// TIA Portal V18 program export: 17 tag tables, 0 data types, 18 data blocks, 24 code blocks (in call order from the OBs), 7 instance data blocks

VAR_GLOBAL   // PLC tag table "PLC_Simulation_Tags"
   "1400_FT115_PV" AT %MD100 : Real;   // Lưu lượng dòng liệu đo được tại FT115
   "1400_FT101_PV" AT %MD104 : Real;   // Lưu lượng dòng liệu đo được tại FT101
   "1400_1_02_PV" AT %MD108 : Real;   // Giá trị đo của cảm biến 1-02
   "1406_TX35_PV" AT %MD112 : Real;   // Giá trị đo cảm biến nhiệt độ/áp suất TX35
   "1400_TT64_PV" AT %MD116 : Real;   // Nhiệt độ đo được tại TT64
   "1400_TT32_PV" AT %MD120 : Real;   // Nhiệt độ đo được tại TT32
   "1400_LGFE01_PV" AT %MD124 : Real;   // Mức bồn hoặc lưu lượng đo tại LGFE01
   "1400_FS51_PV" AT %MD128 : Real;   // Giá trị lưu lượng đo được tại FS51
   "1400_FY301_PV" AT %MD132 : Real;   // Mức cân hoặc vị trí điều khiển bồn FY301
   "1400_TT101_PV" AT %MD136 : Real;   // Nhiệt độ đo được tại TT101
   "1400_FTT02_PV" AT %MD140 : Real;   // Lưu lượng/nhiệt độ đo được tại FTT02
   "1500S_Trang_Thai" AT %M200.0 : Bool;   // Trạng thái hoạt động dòng liệu 1500S (0: Không chảy, 1: Đang chảy)
   "1404T_Trang_Thai" AT %M200.1 : Bool;   // Trạng thái hoạt động dòng liệu 1404T
   CR_2013_FO_104_Trang_Thai AT %M200.2 : Bool;   // Trạng thái hoạt động dòng liệu CR-2013-FO-104
   BFOC_SS_20_06_Trang_Thai AT %M200.3 : Bool;   // Trạng thái hoạt động dòng liệu BFOC-SS-20-06
   PC03010T01_Trang_Thai AT %M200.4 : Bool;   // Trạng thái dòng liệu đầu ra PC03010T01
   "1401_Trang_Thai" AT %M200.5 : Bool;   // Trạng thái dòng liệu xả đáy 1401
   "1400_PT91_Chay" AT %M200.6 : Bool;   // Tín hiệu báo chạy bơm 1400PT91 (1: Chạy)
   "1400_KCK01_Chay" AT %M200.7 : Bool;   // Tín hiệu báo chạy cánh khuấy bồn 1400KCK01
   "1400_FT102_Mo" AT %M201.0 : Bool;   // Tín hiệu báo mở van nạp liệu 1400FT102
   "1400_TY33_Mo" AT %M201.1 : Bool;   // Tín hiệu báo mở van điều khiển cooling 1400TY33
   "160_FEC53_Mo" AT %M201.2 : Bool;   // Tín hiệu báo mở van kẹp 160 FEC53
   "1400_TXC32_Mo" AT %M201.3 : Bool;   // Tín hiệu báo mở van điều khiển 1400TXC32
   "1400_TC32_Mo" AT %M201.4 : Bool;   // Tín hiệu báo mở van điều khiển 1400TC32
   "1400_FIC01_Mo" AT %M201.5 : Bool;   // Tín hiệu báo mở van điều khiển 1400FIC01
   "1400_FS51_Mo" AT %M201.6 : Bool;   // Tín hiệu báo mở van xả đáy 1400FS51
   "1500S_Status" AT %MW300 : Int;   // Mã trạng thái dòng liệu 1500S (0: Dừng, 1: Chạy, 2: Lỗi)
   "1404T_Status" AT %MW302 : Int;   // Mã trạng thái dòng liệu 1404T
   CR_2013_FO_104_Status AT %MW304 : Int;   // Mã trạng thái dòng liệu CR-2013-FO-104
   BFOC_SS_20_06_Status AT %MW306 : Int;   // Mã trạng thái dòng liệu BFOC-SS-20-06
   PC03010T01_Status AT %MW308 : Int;   // Mã trạng thái dòng liệu PC03010T01
   "1401_Status" AT %MW310 : Int;   // Mã trạng thái dòng liệu xả đáy 1401
   "1400_PT91_Status" AT %MW312 : Int;   // Mã trạng thái hoạt động bơm 1400PT91 (0: Dừng, 1: Chạy, 2: Lỗi)
   "1400_KCK01_Status" AT %MW314 : Int;   // Mã trạng thái hoạt động cánh khuấy 1400KCK01
   "1400_FT102_Status" AT %MW316 : Int;   // Mã trạng thái hoạt động van 1400FT102 (0: Đóng, 1: Mở, 2: Lỗi)
   "1400_TY33_Status" AT %MW318 : Int;   // Mã trạng thái hoạt động van 1400TY33
   "160_FEC53_Status" AT %MW320 : Int;   // Mã trạng thái hoạt động van 160 FEC53
   "1400_TXC32_Status" AT %MW322 : Int;   // Mã trạng thái hoạt động van 1400TXC32
   "1400_TC32_Status" AT %MW324 : Int;   // Mã trạng thái hoạt động van 1400TC32
   "1400_FIC01_Status" AT %MW326 : Int;   // Mã trạng thái hoạt động van 1400FIC01
   "1400_FS51_Status" AT %MW328 : Int;   // Mã trạng thái hoạt động van 1400FS51
   Sim_Counter AT %MD400 : Real;   // Biến đếm trung gian cho sóng tam giác mô phỏng
   Sim_Dir AT %M404.0 : Bool;   // Bit hướng đếm mô phỏng (0: Tăng, 1: Giảm)
   Sim_Val_Norm AT %MD408 : Real;   // Giá trị đếm đã chuẩn hóa về dải 0.0 - 1.0
   Timer_Sim_Pulse_Output AT %M404.1 : Bool;   // Xung kích hoạt đếm từ Timer
END_VAR

VAR_GLOBAL   // PLC tag table "AI_Tags"
   AI_Nut_Khoi_Dong AT %I0.0 : Bool;   // Nút khởi động vật lý
   AI_Nut_Khoi_Dong_HMI AT %M110.0 : Bool;   // Tín hiệu mô phỏng/HMI song song cho Nút khởi động vật lý
   AI_Nut_Khoi_Dong_HMI_Gated AT %M320.0 : Bool;   // Tín hiệu HMI đã qua xử lý chế độ cho Nút khởi động vật lý
   AI_Nut_Khoi_Dong_Eff AT %M320.1 : Bool;   // Tín hiệu thực tế/mô phỏng hiệu dụng cho Nút khởi động vật lý
   AI_Nut_Dung AT %I0.1 : Bool;   // Nút dừng vật lý
   AI_Nut_Dung_HMI AT %M110.1 : Bool;   // Tín hiệu mô phỏng/HMI song song cho Nút dừng vật lý
   AI_Nut_Dung_HMI_Gated AT %M320.2 : Bool;   // Tín hiệu HMI đã qua xử lý chế độ cho Nút dừng vật lý
   AI_Nut_Dung_Eff AT %M320.3 : Bool;   // Tín hiệu thực tế/mô phỏng hiệu dụng cho Nút dừng vật lý
   AI_Nut_Reset AT %I0.2 : Bool;   // Nút reset lỗi vật lý
   AI_Nut_Reset_HMI AT %M110.2 : Bool;   // Tín hiệu mô phỏng/HMI song song cho Nút reset lỗi vật lý
   AI_Nut_Reset_HMI_Gated AT %M320.4 : Bool;   // Tín hiệu HMI đã qua xử lý chế độ cho Nút reset lỗi vật lý
   AI_Nut_Reset_Eff AT %M320.5 : Bool;   // Tín hiệu thực tế/mô phỏng hiệu dụng cho Nút reset lỗi vật lý
   AI_Nut_EStop AT %I0.3 : Bool;   // Nút dừng khẩn vật lý
   AI_Nut_EStop_HMI AT %M110.3 : Bool;   // Tín hiệu mô phỏng/HMI song song cho Nút dừng khẩn vật lý
   AI_Nut_EStop_HMI_Gated AT %M320.6 : Bool;   // Tín hiệu HMI đã qua xử lý chế độ cho Nút dừng khẩn vật lý
   AI_Nut_EStop_Eff AT %M320.7 : Bool;   // Tín hiệu thực tế/mô phỏng hiệu dụng cho Nút dừng khẩn vật lý
   AI_FT3200_Bon1 AT %ID100 : Real;   // Cảm biến lưu lượng nước dosing vào Bồn 1
   AI_FT3200_Bon1_HMI AT %MD700 : Real;   // Giá trị mô phỏng/HMI song song cho Cảm biến lưu lượng nước dosing vào Bồn 1
   AI_FT3200_Bon1_Use_HMI AT %M420.0 : Bool;   // Chọn chế độ mô phỏng HMI cho Cảm biến lưu lượng nước dosing vào Bồn 1
   AI_FT3200_Bon1_Sim_Req AT %M321.0 : Bool;   // Yêu cầu mô phỏng cảm biến cho Cảm biến lưu lượng nước dosing vào Bồn 1
   AI_FT3200_Bon1_Sim_Active AT %M321.1 : Bool;   // Mô phỏng cảm biến đang hoạt động cho Cảm biến lưu lượng nước dosing vào Bồn 1
   AI_FT3200_Bon1_Eff AT %MD704 : Real;   // Giá trị thực tế/mô phỏng hiệu dụng cho Cảm biến lưu lượng nước dosing vào Bồn 1
   AI_FQ3200_Bon1 AT %ID104 : Real;   // Bộ đếm lưu lượng tích lũy Bồn 1
   AI_FQ3200_Bon1_HMI AT %MD708 : Real;   // Giá trị mô phỏng/HMI song song cho Bộ đếm lưu lượng tích lũy Bồn 1
   AI_FQ3200_Bon1_Use_HMI AT %M420.1 : Bool;   // Chọn chế độ mô phỏng HMI cho Bộ đếm lưu lượng tích lũy Bồn 1
   AI_FQ3200_Bon1_Sim_Req AT %M321.2 : Bool;   // Yêu cầu mô phỏng cảm biến cho Bộ đếm lưu lượng tích lũy Bồn 1
   AI_FQ3200_Bon1_Sim_Active AT %M321.3 : Bool;   // Mô phỏng cảm biến đang hoạt động cho Bộ đếm lưu lượng tích lũy Bồn 1
   AI_FQ3200_Bon1_Eff AT %MD712 : Real;   // Giá trị thực tế/mô phỏng hiệu dụng cho Bộ đếm lưu lượng tích lũy Bồn 1
   AI_LS3202_Bon1_Cao AT %I0.4 : Bool;   // Cảm biến mức cao Bồn 1
   AI_LS3202_Bon1_Cao_HMI AT %M110.4 : Bool;   // Tín hiệu mô phỏng/HMI song song cho Cảm biến mức cao Bồn 1
   AI_LS3202_Bon1_Cao_HMI_Gated AT %M321.4 : Bool;   // Tín hiệu HMI đã qua xử lý chế độ cho Cảm biến mức cao Bồn 1
   AI_LS3202_Bon1_Cao_Eff AT %M321.5 : Bool;   // Tín hiệu thực tế/mô phỏng hiệu dụng cho Cảm biến mức cao Bồn 1
   AI_LT3203_Bon1 AT %ID108 : Real;   // Cảm biến mức liên tục Bồn 1
   AI_LT3203_Bon1_HMI AT %MD716 : Real;   // Giá trị mô phỏng/HMI song song cho Cảm biến mức liên tục Bồn 1
   AI_LT3203_Bon1_Use_HMI AT %M420.2 : Bool;   // Chọn chế độ mô phỏng HMI cho Cảm biến mức liên tục Bồn 1
   AI_LT3203_Bon1_Sim_Req AT %M321.6 : Bool;   // Yêu cầu mô phỏng cảm biến cho Cảm biến mức liên tục Bồn 1
   AI_LT3203_Bon1_Sim_Active AT %M321.7 : Bool;   // Mô phỏng cảm biến đang hoạt động cho Cảm biến mức liên tục Bồn 1
   AI_LT3203_Bon1_Eff AT %MD720 : Real;   // Giá trị thực tế/mô phỏng hiệu dụng cho Cảm biến mức liên tục Bồn 1
   AI_TT3204_Bon1 AT %ID112 : Real;   // Cảm biến nhiệt độ Bồn 1
   AI_TT3204_Bon1_HMI AT %MD724 : Real;   // Giá trị mô phỏng/HMI song song cho Cảm biến nhiệt độ Bồn 1
   AI_TT3204_Bon1_Use_HMI AT %M420.3 : Bool;   // Chọn chế độ mô phỏng HMI cho Cảm biến nhiệt độ Bồn 1
   AI_TT3204_Bon1_Sim_Req AT %M322.0 : Bool;   // Yêu cầu mô phỏng cảm biến cho Cảm biến nhiệt độ Bồn 1
   AI_TT3204_Bon1_Sim_Active AT %M322.1 : Bool;   // Mô phỏng cảm biến đang hoạt động cho Cảm biến nhiệt độ Bồn 1
   AI_TT3204_Bon1_Eff AT %MD728 : Real;   // Giá trị thực tế/mô phỏng hiệu dụng cho Cảm biến nhiệt độ Bồn 1
   AI_FT3205_Bon2 AT %ID116 : Real;   // Cảm biến lưu lượng nước dosing vào Bồn 2
   AI_FT3205_Bon2_HMI AT %MD732 : Real;   // Giá trị mô phỏng/HMI song song cho Cảm biến lưu lượng nước dosing vào Bồn 2
   AI_FT3205_Bon2_Use_HMI AT %M420.4 : Bool;   // Chọn chế độ mô phỏng HMI cho Cảm biến lưu lượng nước dosing vào Bồn 2
   AI_FT3205_Bon2_Sim_Req AT %M322.2 : Bool;   // Yêu cầu mô phỏng cảm biến cho Cảm biến lưu lượng nước dosing vào Bồn 2
   AI_FT3205_Bon2_Sim_Active AT %M322.3 : Bool;   // Mô phỏng cảm biến đang hoạt động cho Cảm biến lưu lượng nước dosing vào Bồn 2
   AI_FT3205_Bon2_Eff AT %MD736 : Real;   // Giá trị thực tế/mô phỏng hiệu dụng cho Cảm biến lưu lượng nước dosing vào Bồn 2
   AI_FQ3205_Bon2 AT %ID120 : Real;   // Bộ đếm lưu lượng tích lũy Bồn 2
   AI_FQ3205_Bon2_HMI AT %MD740 : Real;   // Giá trị mô phỏng/HMI song song cho Bộ đếm lưu lượng tích lũy Bồn 2
   AI_FQ3205_Bon2_Use_HMI AT %M420.5 : Bool;   // Chọn chế độ mô phỏng HMI cho Bộ đếm lưu lượng tích lũy Bồn 2
   AI_FQ3205_Bon2_Sim_Req AT %M322.4 : Bool;   // Yêu cầu mô phỏng cảm biến cho Bộ đếm lưu lượng tích lũy Bồn 2
   AI_FQ3205_Bon2_Sim_Active AT %M322.5 : Bool;   // Mô phỏng cảm biến đang hoạt động cho Bộ đếm lưu lượng tích lũy Bồn 2
   AI_FQ3205_Bon2_Eff AT %MD744 : Real;   // Giá trị thực tế/mô phỏng hiệu dụng cho Bộ đếm lưu lượng tích lũy Bồn 2
   AI_LT3209_Bon2 AT %ID124 : Real;   // Cảm biến mức liên tục Bồn 2
   AI_LT3209_Bon2_HMI AT %MD748 : Real;   // Giá trị mô phỏng/HMI song song cho Cảm biến mức liên tục Bồn 2
   AI_LT3209_Bon2_Use_HMI AT %M420.6 : Bool;   // Chọn chế độ mô phỏng HMI cho Cảm biến mức liên tục Bồn 2
   AI_LT3209_Bon2_Sim_Req AT %M322.6 : Bool;   // Yêu cầu mô phỏng cảm biến cho Cảm biến mức liên tục Bồn 2
   AI_LT3209_Bon2_Sim_Active AT %M322.7 : Bool;   // Mô phỏng cảm biến đang hoạt động cho Cảm biến mức liên tục Bồn 2
   AI_LT3209_Bon2_Eff AT %MD752 : Real;   // Giá trị thực tế/mô phỏng hiệu dụng cho Cảm biến mức liên tục Bồn 2
   AI_TT3208_Bon2 AT %ID128 : Real;   // Cảm biến nhiệt độ Bồn 2
   AI_TT3208_Bon2_HMI AT %MD756 : Real;   // Giá trị mô phỏng/HMI song song cho Cảm biến nhiệt độ Bồn 2
   AI_TT3208_Bon2_Use_HMI AT %M420.7 : Bool;   // Chọn chế độ mô phỏng HMI cho Cảm biến nhiệt độ Bồn 2
   AI_TT3208_Bon2_Sim_Req AT %M323.0 : Bool;   // Yêu cầu mô phỏng cảm biến cho Cảm biến nhiệt độ Bồn 2
   AI_TT3208_Bon2_Sim_Active AT %M323.1 : Bool;   // Mô phỏng cảm biến đang hoạt động cho Cảm biến nhiệt độ Bồn 2
   AI_TT3208_Bon2_Eff AT %MD760 : Real;   // Giá trị thực tế/mô phỏng hiệu dụng cho Cảm biến nhiệt độ Bồn 2
   AI_V3230_Nuoc_Bon1 AT %Q0.0 : Bool;   // Van on/off cấp nước Bồn 1
   AI_V3230_Nuoc_Bon1_M AT %M220.0 : Bool;   // Tag gương phản hồi HMI cho Van on/off cấp nước Bồn 1
   AI_CV3201_Nuoc_Bon1 AT %QD100 : Real;   // Van tuyến tính cấp nước Bồn 1
   AI_CV3201_Nuoc_Bon1_M AT %MD1200 : Real;   // Tag gương phản hồi HMI cho Van tuyến tính cấp nước Bồn 1
   AI_AGTR3260_Khuay_Bon1 AT %Q0.1 : Bool;   // Động cơ khuấy Bồn 1
   AI_AGTR3260_Khuay_Bon1_M AT %M220.1 : Bool;   // Tag gương phản hồi HMI cho Động cơ khuấy Bồn 1
   AI_AGTR3260_Toc_Do_AO AT %QD104 : Real;   // Tín hiệu tốc độ khuấy Bồn 1
   AI_AGTR3260_Toc_Do_AO_M AT %MD1204 : Real;   // Tag gương phản hồi HMI cho Tín hiệu tốc độ khuấy Bồn 1
   AI_V3232_Xa_Bon1 AT %Q0.2 : Bool;   // Van xả đáy Bồn 1 số 1
   AI_V3232_Xa_Bon1_M AT %M220.2 : Bool;   // Tag gương phản hồi HMI cho Van xả đáy Bồn 1 số 1
   AI_V3233_Xa_Bon1 AT %Q0.3 : Bool;   // Van xả đáy Bồn 1 số 2
   AI_V3233_Xa_Bon1_M AT %M220.3 : Bool;   // Tag gương phản hồi HMI cho Van xả đáy Bồn 1 số 2
   AI_V3234_Xa_Bon1 AT %Q0.4 : Bool;   // Van xả đáy Bồn 1 số 3
   AI_V3234_Xa_Bon1_M AT %M220.4 : Bool;   // Tag gương phản hồi HMI cho Van xả đáy Bồn 1 số 3
   AI_V3235_Nuoc_Bon2 AT %Q0.5 : Bool;   // Van on/off cấp nước Bồn 2
   AI_V3235_Nuoc_Bon2_M AT %M220.5 : Bool;   // Tag gương phản hồi HMI cho Van on/off cấp nước Bồn 2
   AI_CV3206_Hoi_Bon2 AT %QD108 : Real;   // Van hơi/nhiệt Bồn 2 ở chế độ cho phép
   AI_CV3206_Hoi_Bon2_M AT %MD1208 : Real;   // Tag gương phản hồi HMI cho Van hơi/nhiệt Bồn 2 ở chế độ cho phép
   AI_VFD_Bon2_Run AT %Q0.6 : Bool;   // Lệnh chạy VFD động cơ Bồn 2
   AI_VFD_Bon2_Run_M AT %M220.6 : Bool;   // Tag gương phản hồi HMI cho Lệnh chạy VFD động cơ Bồn 2
   AI_VFD_Bon2_Dao_Chieu AT %Q0.7 : Bool;   // Lệnh đảo chiều VFD động cơ Bồn 2
   AI_VFD_Bon2_Dao_Chieu_M AT %M220.7 : Bool;   // Tag gương phản hồi HMI cho Lệnh đảo chiều VFD động cơ Bồn 2
   AI_VFD_Bon2_Toc_Do_AO AT %QD112 : Real;   // Tốc độ đặt VFD Bồn 2 từ HMI setpoint
   AI_VFD_Bon2_Toc_Do_AO_M AT %MD1212 : Real;   // Tag gương phản hồi HMI cho Tốc độ đặt VFD Bồn 2 từ HMI setpoint
   AI_V3237_Xa_Bon2 AT %Q1.0 : Bool;   // Van xả đáy Bồn 2 số 1
   AI_V3237_Xa_Bon2_M AT %M221.0 : Bool;   // Tag gương phản hồi HMI cho Van xả đáy Bồn 2 số 1
   AI_V3238_Xa_Bon2 AT %Q1.1 : Bool;   // Van xả đáy Bồn 2 số 2
   AI_V3238_Xa_Bon2_M AT %M221.1 : Bool;   // Tag gương phản hồi HMI cho Van xả đáy Bồn 2 số 2
   AI_V3239_Xa_Bon2 AT %Q1.2 : Bool;   // Van xả đáy Bồn 2 số 3
   AI_V3239_Xa_Bon2_M AT %M221.2 : Bool;   // Tag gương phản hồi HMI cho Van xả đáy Bồn 2 số 3
   AI_Pump3264_Chuyen_Nhanh1 AT %Q1.3 : Bool;   // Bơm chuyển dung dịch Nhánh 1 xuống bồn chứa
   AI_Pump3264_Chuyen_Nhanh1_M AT %M221.3 : Bool;   // Tag gương phản hồi HMI cho Bơm chuyển dung dịch Nhánh 1 xuống bồn chứa
   AI_LT3302_BonChua1 AT %ID164 : Real;   // Cảm biến mức liên tục Bồn chứa 01
   AI_LT3302_BonChua1_HMI AT %MD828 : Real;   // Giá trị mô phỏng/HMI song song cho Cảm biến mức liên tục Bồn chứa 01
   AI_LT3302_BonChua1_Use_HMI AT %M422.0 : Bool;   // Chọn chế độ mô phỏng HMI cho Cảm biến mức liên tục Bồn chứa 01
   AI_LT3302_BonChua1_Sim_Req AT %M325.4 : Bool;   // Yêu cầu mô phỏng cảm biến cho Cảm biến mức liên tục Bồn chứa 01
   AI_LT3302_BonChua1_Sim_Active AT %M325.5 : Bool;   // Mô phỏng cảm biến đang hoạt động cho Cảm biến mức liên tục Bồn chứa 01
   AI_LT3302_BonChua1_Eff AT %MD832 : Real;   // Giá trị thực tế/mô phỏng hiệu dụng cho Cảm biến mức liên tục Bồn chứa 01
   AI_TT3301_BonChua1 AT %ID168 : Real;   // Cảm biến nhiệt độ Bồn chứa 01
   AI_TT3301_BonChua1_HMI AT %MD836 : Real;   // Giá trị mô phỏng/HMI song song cho Cảm biến nhiệt độ Bồn chứa 01
   AI_TT3301_BonChua1_Use_HMI AT %M422.1 : Bool;   // Chọn chế độ mô phỏng HMI cho Cảm biến nhiệt độ Bồn chứa 01
   AI_TT3301_BonChua1_Sim_Req AT %M325.6 : Bool;   // Yêu cầu mô phỏng cảm biến cho Cảm biến nhiệt độ Bồn chứa 01
   AI_TT3301_BonChua1_Sim_Active AT %M325.7 : Bool;   // Mô phỏng cảm biến đang hoạt động cho Cảm biến nhiệt độ Bồn chứa 01
   AI_TT3301_BonChua1_Eff AT %MD840 : Real;   // Giá trị thực tế/mô phỏng hiệu dụng cho Cảm biến nhiệt độ Bồn chứa 01
   AI_TT3303_TraoDoiNhiet AT %ID172 : Real;   // Cảm biến nhiệt độ bộ trao đổi nhiệt
   AI_TT3303_TraoDoiNhiet_HMI AT %MD844 : Real;   // Giá trị mô phỏng/HMI song song cho Cảm biến nhiệt độ bộ trao đổi nhiệt
   AI_TT3303_TraoDoiNhiet_Use_HMI AT %M422.2 : Bool;   // Chọn chế độ mô phỏng HMI cho Cảm biến nhiệt độ bộ trao đổi nhiệt
   AI_TT3303_TraoDoiNhiet_Sim_Req AT %M326.0 : Bool;   // Yêu cầu mô phỏng cảm biến cho Cảm biến nhiệt độ bộ trao đổi nhiệt
   AI_TT3303_TraoDoiNhiet_Sim_Active AT %M326.1 : Bool;   // Mô phỏng cảm biến đang hoạt động cho Cảm biến nhiệt độ bộ trao đổi nhiệt
   AI_TT3303_TraoDoiNhiet_Eff AT %MD848 : Real;   // Giá trị thực tế/mô phỏng hiệu dụng cho Cảm biến nhiệt độ bộ trao đổi nhiệt
   AI_LT3307_BonChua2 AT %ID176 : Real;   // Cảm biến mức liên tục Bồn chứa 02
   AI_LT3307_BonChua2_HMI AT %MD852 : Real;   // Giá trị mô phỏng/HMI song song cho Cảm biến mức liên tục Bồn chứa 02
   AI_LT3307_BonChua2_Use_HMI AT %M422.3 : Bool;   // Chọn chế độ mô phỏng HMI cho Cảm biến mức liên tục Bồn chứa 02
   AI_LT3307_BonChua2_Sim_Req AT %M326.2 : Bool;   // Yêu cầu mô phỏng cảm biến cho Cảm biến mức liên tục Bồn chứa 02
   AI_LT3307_BonChua2_Sim_Active AT %M326.3 : Bool;   // Mô phỏng cảm biến đang hoạt động cho Cảm biến mức liên tục Bồn chứa 02
   AI_LT3307_BonChua2_Eff AT %MD856 : Real;   // Giá trị thực tế/mô phỏng hiệu dụng cho Cảm biến mức liên tục Bồn chứa 02
   AI_TT3306_BonChua2 AT %ID180 : Real;   // Cảm biến nhiệt độ Bồn chứa 02
   AI_TT3306_BonChua2_HMI AT %MD860 : Real;   // Giá trị mô phỏng/HMI song song cho Cảm biến nhiệt độ Bồn chứa 02
   AI_TT3306_BonChua2_Use_HMI AT %M422.4 : Bool;   // Chọn chế độ mô phỏng HMI cho Cảm biến nhiệt độ Bồn chứa 02
   AI_TT3306_BonChua2_Sim_Req AT %M326.4 : Bool;   // Yêu cầu mô phỏng cảm biến cho Cảm biến nhiệt độ Bồn chứa 02
   AI_TT3306_BonChua2_Sim_Active AT %M326.5 : Bool;   // Mô phỏng cảm biến đang hoạt động cho Cảm biến nhiệt độ Bồn chứa 02
   AI_TT3306_BonChua2_Eff AT %MD864 : Real;   // Giá trị thực tế/mô phỏng hiệu dụng cho Cảm biến nhiệt độ Bồn chứa 02
   AI_PI3308_Truoc_Filter AT %ID184 : Real;   // Cảm biến áp suất trước màng lọc
   AI_PI3308_Truoc_Filter_HMI AT %MD868 : Real;   // Giá trị mô phỏng/HMI song song cho Cảm biến áp suất trước màng lọc
   AI_PI3308_Truoc_Filter_Use_HMI AT %M422.5 : Bool;   // Chọn chế độ mô phỏng HMI cho Cảm biến áp suất trước màng lọc
   AI_PI3308_Truoc_Filter_Sim_Req AT %M326.6 : Bool;   // Yêu cầu mô phỏng cảm biến cho Cảm biến áp suất trước màng lọc
   AI_PI3308_Truoc_Filter_Sim_Active AT %M326.7 : Bool;   // Mô phỏng cảm biến đang hoạt động cho Cảm biến áp suất trước màng lọc
   AI_PI3308_Truoc_Filter_Eff AT %MD872 : Real;   // Giá trị thực tế/mô phỏng hiệu dụng cho Cảm biến áp suất trước màng lọc
   AI_FT3309_Xa_Thanh_Pham AT %ID188 : Real;   // Cảm biến lưu lượng xả thành phẩm
   AI_FT3309_Xa_Thanh_Pham_HMI AT %MD876 : Real;   // Giá trị mô phỏng/HMI song song cho Cảm biến lưu lượng xả thành phẩm
   AI_FT3309_Xa_Thanh_Pham_Use_HMI AT %M422.6 : Bool;   // Chọn chế độ mô phỏng HMI cho Cảm biến lưu lượng xả thành phẩm
   AI_FT3309_Xa_Thanh_Pham_Sim_Req AT %M327.0 : Bool;   // Yêu cầu mô phỏng cảm biến cho Cảm biến lưu lượng xả thành phẩm
   AI_FT3309_Xa_Thanh_Pham_Sim_Active AT %M327.1 : Bool;   // Mô phỏng cảm biến đang hoạt động cho Cảm biến lưu lượng xả thành phẩm
   AI_FT3309_Xa_Thanh_Pham_Eff AT %MD880 : Real;   // Giá trị thực tế/mô phỏng hiệu dụng cho Cảm biến lưu lượng xả thành phẩm
   AI_LSH3310_Pheu_Cao AT %I0.6 : Bool;   // Cảm biến mức cao phễu chiết rót
   AI_LSH3310_Pheu_Cao_HMI AT %M110.6 : Bool;   // Tín hiệu mô phỏng/HMI song song cho Cảm biến mức cao phễu chiết rót
   AI_LSH3310_Pheu_Cao_HMI_Gated AT %M327.2 : Bool;   // Tín hiệu HMI đã qua xử lý chế độ cho Cảm biến mức cao phễu chiết rót
   AI_LSH3310_Pheu_Cao_Eff AT %M327.3 : Bool;   // Tín hiệu thực tế/mô phỏng hiệu dụng cho Cảm biến mức cao phễu chiết rót
   AI_LSL3311_Pheu_Thap AT %I0.7 : Bool;   // Cảm biến mức thấp phễu chiết rót
   AI_LSL3311_Pheu_Thap_HMI AT %M110.7 : Bool;   // Tín hiệu mô phỏng/HMI song song cho Cảm biến mức thấp phễu chiết rót
   AI_LSL3311_Pheu_Thap_HMI_Gated AT %M327.4 : Bool;   // Tín hiệu HMI đã qua xử lý chế độ cho Cảm biến mức thấp phễu chiết rót
   AI_LSL3311_Pheu_Thap_Eff AT %M327.5 : Bool;   // Tín hiệu thực tế/mô phỏng hiệu dụng cho Cảm biến mức thấp phễu chiết rót
   AI_V3331_Xa_BonChua1 AT %Q3.0 : Bool;   // Van xả đáy Bồn chứa 01 số 1
   AI_V3331_Xa_BonChua1_M AT %M223.0 : Bool;   // Tag gương phản hồi HMI cho Van xả đáy Bồn chứa 01 số 1
   AI_V3332_Xa_BonChua1 AT %Q3.1 : Bool;   // Van xả đáy Bồn chứa 01 số 2
   AI_V3332_Xa_BonChua1_M AT %M223.1 : Bool;   // Tag gương phản hồi HMI cho Van xả đáy Bồn chứa 01 số 2
   AI_Pump3361_LuanChuyen_BonChua1 AT %Q3.2 : Bool;   // Bơm luân chuyển Bồn chứa 01
   AI_Pump3361_LuanChuyen_BonChua1_M AT %M223.2 : Bool;   // Tag gương phản hồi HMI cho Bơm luân chuyển Bồn chứa 01
   AI_Pump3362_Xa_BonChua1 AT %Q3.3 : Bool;   // Bơm xả Bồn chứa 01
   AI_Pump3362_Xa_BonChua1_M AT %M223.3 : Bool;   // Tag gương phản hồi HMI cho Bơm xả Bồn chứa 01
   AI_V3333_DieuHuong_BonChua1 AT %Q3.4 : Bool;   // Van điều hướng Bồn chứa 01 số 1
   AI_V3333_DieuHuong_BonChua1_M AT %M223.4 : Bool;   // Tag gương phản hồi HMI cho Van điều hướng Bồn chứa 01 số 1
   AI_V3334_DieuHuong_BonChua1 AT %Q3.5 : Bool;   // Van điều hướng Bồn chứa 01 số 2
   AI_V3334_DieuHuong_BonChua1_M AT %M223.5 : Bool;   // Tag gương phản hồi HMI cho Van điều hướng Bồn chứa 01 số 2
   AI_V3335_DieuHuong_BonChua1 AT %Q3.6 : Bool;   // Van điều hướng Bồn chứa 01 số 3
   AI_V3335_DieuHuong_BonChua1_M AT %M223.6 : Bool;   // Tag gương phản hồi HMI cho Van điều hướng Bồn chứa 01 số 3
   AI_CV3304_Nuoc_Lam_Mat AT %QD132 : Real;   // Van tuyến tính nước làm mát
   AI_CV3304_Nuoc_Lam_Mat_M AT %MD1232 : Real;   // Tag gương phản hồi HMI cho Van tuyến tính nước làm mát
   AI_V3338_Xa_BonChua2 AT %Q3.7 : Bool;   // Van xả đáy Bồn chứa 02 số 1
   AI_V3338_Xa_BonChua2_M AT %M223.7 : Bool;   // Tag gương phản hồi HMI cho Van xả đáy Bồn chứa 02 số 1
   AI_V3339_Xa_BonChua2 AT %Q4.0 : Bool;   // Van xả đáy Bồn chứa 02 số 2
   AI_V3339_Xa_BonChua2_M AT %M224.0 : Bool;   // Tag gương phản hồi HMI cho Van xả đáy Bồn chứa 02 số 2
   AI_Pump3364_Filter AT %Q4.1 : Bool;   // Bơm qua màng lọc CCP số 1
   AI_Pump3364_Filter_M AT %M224.1 : Bool;   // Tag gương phản hồi HMI cho Bơm qua màng lọc CCP số 1
   AI_Pump3365_Filter AT %Q4.2 : Bool;   // Bơm qua màng lọc CCP số 2
   AI_Pump3365_Filter_M AT %M224.2 : Bool;   // Tag gương phản hồi HMI cho Bơm qua màng lọc CCP số 2
   AI_V3340_Duong_Filter AT %Q4.3 : Bool;   // Van đường ống Filter số 1
   AI_V3340_Duong_Filter_M AT %M224.3 : Bool;   // Tag gương phản hồi HMI cho Van đường ống Filter số 1
   AI_V3341_Duong_Filter AT %Q4.4 : Bool;   // Van đường ống Filter số 2
   AI_V3341_Duong_Filter_M AT %M224.4 : Bool;   // Tag gương phản hồi HMI cho Van đường ống Filter số 2
   AI_CV_Filler_Cap_Dich AT %QD136 : Real;   // Van tuyến tính cấp dịch xuống phễu chiết rót
   AI_CV_Filler_Cap_Dich_M AT %MD1236 : Real;   // Tag gương phản hồi HMI cho Van tuyến tính cấp dịch xuống phễu chiết rót
   AI_Coi_Bao_Dong AT %Q4.5 : Bool;   // Còi báo động chung
   AI_Coi_Bao_Dong_M AT %M224.5 : Bool;   // Tag gương phản hồi HMI cho Còi báo động chung
   AI_HMI_Operator_Login AT %M422.7 : Bool;   // Đăng nhập quyền Operator
   AI_HMI_Engineer_Login AT %M423.0 : Bool;   // Đăng nhập quyền Engineer
   AI_HMI_Admin_Login AT %M423.1 : Bool;   // Đăng nhập quyền Admin
   AI_HMI_Che_Do_Manual AT %M423.2 : Bool;   // Cho phép điều khiển tay từng thiết bị
   AI_HMI_Ack_Alarm AT %M423.3 : Bool;   // Xác nhận cảnh báo
   AI_HMI_Reset_Alarm AT %M423.4 : Bool;   // Reset alarm bằng HMI
   AI_Gia_Lap_Mat_Ket_Noi_HMI AT %M423.5 : Bool;   // Nút giả lập mất kết nối PLC
   AI_HMI_User_Level AT %MW520 : Int;   // Mức quyền hiện tại: 1 Operator, 2 Engineer, 3 Admin
   AI_HMI_Cho_Phep_Sua_Thong_So AT %M327.6 : Bool;   // Cờ cho phép sửa công thức và PID
   AI_HMI_Alarm_Status AT %MW522 : Int;   // Mã cảnh báo tổng hợp cho WinCC TextList
   AI_HMI_AnToan_Status AT %MW524 : Int;   // Mã chẩn đoán an toàn ưu tiên
   AI_PLC1_Auto_Enable AT %M327.7 : Bool;   // Cho phép chạy Auto Nhánh 1 Bồn 1-2
   AI_PLC1_EStop_Latch AT %M328.0 : Bool;   // Chốt dừng khẩn HMI/SCADA Nhánh 1 Bồn 1-2
   AI_PLC1_Loi_Tong AT %M328.1 : Bool;   // Lỗi tổng khóa Auto Nhánh 1 Bồn 1-2
   AI_PLC1_Loi_Dry_Run AT %M328.2 : Bool;   // Lỗi chạy khô bơm Nhánh 1 Bồn 1-2
   AI_PLC1_Loi_Dosing AT %M328.3 : Bool;   // Lỗi quá thời gian dosing Nhánh 1 Bồn 1-2
   AI_PLC1_Loi_Truyen_Thong AT %M328.4 : Bool;   // Lỗi truyền thông mô phỏng Nhánh 1 Bồn 1-2
   AI_PLC1_State AT %MW526 : Int;   // Mã bước chu trình Nhánh 1 Bồn 1-2
   AI_PLC1_Step_Bon1_Dosing AT %M329.3 : Bool;   // Bồn 1 đang dosing nước
   AI_PLC1_Step_Bon1_Tip AT %M329.4 : Bool;   // Bồn 1 đang mô phỏng tip cốt tương Nhật Bản
   AI_PLC1_Step_Bon1_Khuay AT %M329.5 : Bool;   // Bồn 1 đang khuấy ban đầu
   AI_PLC1_Step_Bon1_Xa AT %M329.6 : Bool;   // Bồn 1 đang xả sang Bồn 2
   AI_PLC1_Step_Bon2_Dosing AT %M329.7 : Bool;   // Bồn 2 đang dosing bổ sung
   AI_PLC1_Step_Bon2_Tip AT %M330.0 : Bool;   // Bồn 2 đang tip phụ gia
   AI_PLC1_Step_Bon2_Khuay_Thuan AT %M330.1 : Bool;   // Bồn 2 khuấy chiều thuận
   AI_PLC1_Step_Bon2_Khuay_Nghich AT %M330.2 : Bool;   // Bồn 2 khuấy chiều ngược
   AI_PLC1_Step_Bon2_PID AT %M330.3 : Bool;   // Bồn 2 gia nhiệt PID
   AI_PLC1_Step_Bon2_Thanh_Trung AT %M330.4 : Bool;   // Bồn 2 giữ thời gian thanh trùng
   AI_PLC1_Me_Nhanh1_Hoan_Thanh AT %M330.5 : Bool;   // Nhánh 1 hoàn thành và sẵn sàng xả xuống bồn chứa
   AI_PLC1_Xa_Bon1_Xong AT %M330.6 : Bool;   // Bồn 1 đã xả hết
   AI_PLC1_Xa_Bon2_Xong AT %M330.7 : Bool;   // Bồn 2 đã xả hết
   AI_BonChua_Step_Nhan_Dich AT %M332.4 : Bool;   // Bồn chứa 01 đang nhận dịch từ nhánh hoàn thành
   AI_BonChua_Step_Giai_Nhiet AT %M332.5 : Bool;   // Bồn chứa 01 đang giải nhiệt xuống 45 độ C
   AI_BonChua_Step_Chuyen_Bon2 AT %M332.6 : Bool;   // Đang chuyển từ Bồn chứa 01 sang Bồn chứa 02
   AI_BonChua_Step_Loc_Chiet AT %M332.7 : Bool;   // Đang lọc CCP và chiết rót
   AI_BonChua_Me_Hoan_Thanh AT %M333.0 : Bool;   // Hoàn thành một mẻ sản xuất chung
   AI_BonChua_State AT %MW530 : Int;   // Mã bước cụm bồn chứa và lọc thành phẩm
   AI_BonChua_Owner_Nhanh1 AT %M333.1 : Bool;   // Mức ưu tiên Nhánh 1 sở hữu bồn chứa
   AI_BonChua_Owner_Nhanh2 AT %M333.2 : Bool;   // Mức ưu tiên Nhánh 2 sở hữu bồn chứa
   AI_PLC2_Me_Nhanh2_Hoan_Thanh_Nhan AT %M333.4 : Bool;   // Cờ PLC1 nhận trạng thái hoàn thành từ PLC2
   AI_PLC2_Me_Nhanh2_Hoan_Thanh_Nhan_HMI AT %M111.0 : Bool;   // Tín hiệu mô phỏng/HMI song song cho cờ PLC1 nhận trạng thái hoàn thành từ PLC2
   AI_PLC2_Xa_Bon4_Xong_Nhan AT %M333.5 : Bool;   // Cờ PLC1 nhận trạng thái xả xong Bồn 4 từ PLC2
   AI_Pump3265_Chuyen_Nhanh2_Cmd AT %M333.6 : Bool;   // Lệnh chạy bơm chuyển Nhánh 2 gửi sang PLC2
   AI_Pump3265_Chuyen_Nhanh2_Cmd_M AT %M224.7 : Bool;   // Tag gương phản hồi HMI cho lệnh chạy bơm chuyển Nhánh 2 gửi sang PLC2
   AI_PID_Bon4_SP_Recv AT %MD884 : Real;   // PID Bồn 4 Setpoint nhận từ PLC2
   AI_PID_Bon4_PV_Recv AT %MD888 : Real;   // PID Bồn 4 Process Value nhận từ PLC2
   AI_PID_Bon4_CV_Recv AT %MD892 : Real;   // PID Bồn 4 Control Value nhận từ PLC2
   AI_PLC2_State_Recv AT %MW532 : Int;   // Trạng thái hoạt động PLC2 nhận từ PLC2
   AI_PLC2_Loi_Tong_Recv AT %M334.0 : Bool;   // Cờ lỗi tổng PLC2 nhận từ PLC2
   AI_VFD_Bon2_iStep AT %MW60 : Int;   // Bước quét tuần tự Modbus VFD Bồn 2
   AI_VFD_Bon2_iStep_Reset AT %M335.5 : Bool;   // Cờ reset bộ đếm bước Modbus VFD Bồn 2
   AI_VFD_Bon2_Step0_Req AT %M335.6 : Bool;   // Yêu cầu bước 0 Modbus VFD Bồn 2
   AI_VFD_Bon2_Step1_Req AT %M335.7 : Bool;   // Yêu cầu bước 1 Modbus VFD Bồn 2
   AI_VFD_Bon2_Step2_Req AT %M336.0 : Bool;   // Yêu cầu bước 2 Modbus VFD Bồn 2
   AI_VFD_Bon2_Step3_Req AT %M336.1 : Bool;   // Yêu cầu bước 3 Modbus VFD Bồn 2
   AI_VFD_Bon2_MB_ControlWord AT %MW40 : Word;   // Control Word gửi VFD Bồn 2
   AI_VFD_Bon2_MB_FreqSetpoint AT %MW42 : Int;   // Frequency Setpoint gửi VFD Bồn 2
   AI_VFD_Bon2_MB_StatusWord AT %MW44 : Word;   // Status Word đọc từ VFD Bồn 2
   AI_VFD_Bon2_MB_ActualSpeed AT %MW46 : Int;   // Actual Speed đọc từ VFD Bồn 2
   AI_VFD_Bon2_MB_Error AT %M50.0 : Bool;   // Lỗi Modbus Master VFD Bồn 2
   AI_VFD_Bon2_MB_Busy AT %M50.1 : Bool;   // Modbus Master Busy VFD Bồn 2
   AI_VFD_Bon2_MB_Done AT %M50.2 : Bool;   // Modbus Master Done VFD Bồn 2
   AI_VFD_Bon2_MB_Status AT %MW52 : Word;   // Trạng thái Modbus Master VFD Bồn 2
   AI_VFD_Bon2_MBCL_Done AT %M51.0 : Bool;   // Modbus Comm Load Done VFD Bồn 2
   AI_VFD_Bon2_MBCL_Error AT %M51.1 : Bool;   // Modbus Comm Load Error VFD Bồn 2
   AI_VFD_Bon2_MBCL_Status AT %MW54 : Word;   // Trạng thái Modbus Comm Load VFD Bồn 2
   AI_VFD_Bon2_Freq_Temp AT %MD70 : Real;   // Biến tạm tần số VFD Bồn 2
   AI_VFD_Bon2_Actual_Speed_Feedback AT %MD74 : Real;   // Phản hồi tốc độ thực tế VFD Bồn 2
   AI_VFD_Bon2_Actual_Speed_Feedback_M AT %MD1240 : Real;   // Tag gương phản hồi HMI tốc độ thực tế VFD Bồn 2
   AI_Clock_1Hz AT %M100.5 : Bool;   // Clock 1Hz system memory bit
   AI_FirstScan AT %M101.0 : Bool;   // First Scan system memory bit
   AI_MB_TCP_iStep AT %MW80 : Int;   // Modbus TCP Client step
   AI_MB_TCP_REQ AT %M82.0 : Bool;   // Modbus TCP Client Request
   AI_MB_TCP_DONE AT %M82.2 : Bool;   // Modbus TCP Client Transaction Done
   AI_MB_TCP_ERROR AT %M82.3 : Bool;   // Modbus TCP Client Transaction Error
   AI_MB_TCP_BUSY AT %M82.6 : Bool;   // Modbus TCP Client Transaction Busy
   AI_MB_TCP_STATUS AT %MW84 : Word;   // Modbus TCP Client Status
   AI_MB_TCP_Mode AT %MB88 : USInt;   // Modbus TCP Client Mode
   AI_MB_TCP_DataAddr AT %MD90 : UDInt;   // Modbus TCP Client Data Address
   AI_MB_TCP_DataLen AT %MW94 : UInt;   // Modbus TCP Client Data Length
   AI_Nut_Khoi_Dong_Eff_Old AT %M83.0 : Bool;   // Old value of Start button
   AI_Nut_Khoi_Dong_Eff_Edge AT %M83.6 : Bool;   // Start command edge detected
   AI_Nut_Dung_Eff_Old AT %M83.1 : Bool;   // Old value of Stop button
   AI_Nut_Dung_Eff_Edge AT %M83.7 : Bool;   // Stop command edge detected
   AI_Nut_Reset_Eff_Old AT %M83.2 : Bool;   // Old value of Reset button
   AI_Nut_Reset_Eff_Edge AT %M84.0 : Bool;   // Reset command edge detected
   AI_Nut_EStop_Eff_Old AT %M83.3 : Bool;   // Old value of EStop button
   AI_Nut_EStop_Eff_Edge AT %M84.1 : Bool;   // EStop command edge detected
   AI_Pump3265_Chuyen_Nhanh2_Cmd_Old AT %M83.4 : Bool;   // Old value of Transfer command
   AI_Pump3265_Chuyen_Nhanh2_Cmd_Edge AT %M84.2 : Bool;   // Transfer command edge detected
   AI_PLC1_Load_Default_Cmd_Old AT %M83.5 : Bool;   // Old value of Load Recipe command
   AI_PLC1_Load_Default_Cmd_Edge AT %M84.3 : Bool;   // Load Recipe command edge detected
   AI_MB_TCP_Any_Cmd_Edge AT %M84.4 : Bool;   // Any handshake command edge detected
   AI_PLC1_Tip_Bon1_Xong_HMI AT %M423.6 : Bool;   // Nút mô phỏng tip Bồn 1 đã hoàn tất
   AI_PLC1_Khuay_Bon1_Xong_HMI AT %M423.7 : Bool;   // Nút mô phỏng hết thời gian khuấy Bồn 1
   AI_PLC1_Tip_Bon2_Xong_HMI AT %M424.0 : Bool;   // Nút mô phỏng tip Bồn 2 đã hoàn tất
   AI_PLC1_Khuay_Thuan_Bon2_Xong_HMI AT %M424.1 : Bool;   // Nút mô phỏng hết thời gian khuấy thuận Bồn 2
   AI_PLC1_Khuay_Nghich_Bon2_Xong_HMI AT %M424.2 : Bool;   // Nút mô phỏng hết thời gian khuấy ngược Bồn 2
   AI_PLC1_Thanh_Trung_Bon2_Xong_HMI AT %M424.3 : Bool;   // Nút mô phỏng hết thời gian thanh trùng Bồn 2
   AI_PLC2_Tip_Bon3_Xong_HMI AT %M424.4 : Bool;   // Nút mô phỏng tip Bồn 3 đã hoàn tất
   AI_PLC2_Khuay_Bon3_Xong_HMI AT %M424.5 : Bool;   // Nút mô phỏng hết thời gian khuấy Bồn 3
   AI_PLC2_Tip_Bon4_Xong_HMI AT %M424.6 : Bool;   // Nút mô phỏng tip Bồn 4 đã hoàn tất
   AI_PLC2_Khuay_Thuan_Bon4_Xong_HMI AT %M424.7 : Bool;   // Nút mô phỏng hết thời gian khuấy thuận Bồn 4
   AI_PLC2_Khuay_Nghich_Bon4_Xong_HMI AT %M425.0 : Bool;   // Nút mô phỏng hết thời gian khuấy ngược Bồn 4
   AI_PLC2_Thanh_Trung_Bon4_Xong_HMI AT %M425.1 : Bool;   // Nút mô phỏng hết thời gian thanh trùng Bồn 4
   AI_BonChua_Nhan_Dich_Xong_HMI AT %M425.2 : Bool;   // Nút mô phỏng nhận dịch vào Bồn chứa 01 xong
   AI_BonChua_Chuyen_Bon2_Xong_HMI AT %M425.3 : Bool;   // Nút mô phỏng chuyển sang Bồn chứa 02 xong
   AI_HMI_SP_PLC1_Nuoc_Bon1 AT %MD896 : Real;   // Lượng nước dosing Bồn 1
   AI_HMI_SP_PLC1_Nuoc_Bon2 AT %MD900 : Real;   // Lượng nước dosing bổ sung Bồn 2
   AI_HMI_SP_PLC1_Toc_Do_Bon1 AT %MD904 : Real;   // Tốc độ khuấy Bồn 1
   AI_HMI_SP_PLC1_Toc_Do_Bon2_Main AT %MD908 : Real;   // Tốc độ khuấy chính Bồn 2
   AI_HMI_SP_PLC1_Nhiet_Do_Bon2 AT %MD912 : Real;   // Setpoint nhiệt/PID Bồn 2
   AI_HMI_SP_PLC2_Nuoc_Bon3 AT %MD916 : Real;   // Lượng nước dosing Bồn 3
   AI_HMI_SP_PLC2_Nuoc_Bon4 AT %MD920 : Real;   // Lượng nước dosing bổ sung Bồn 4
   AI_HMI_SP_PLC2_Toc_Do_Bon3 AT %MD924 : Real;   // Tốc độ khuấy Bồn 3
   AI_HMI_SP_PLC2_Toc_Do_Bon4_Main AT %MD928 : Real;   // Tốc độ khuấy chính Bồn 4
   AI_HMI_SP_PLC2_Nhiet_Do_Bon4 AT %MD932 : Real;   // Setpoint nhiệt/PID mô phỏng Bồn 4
   AI_HMI_SP_BonChua1_Nhiet_Giai_Nhiet AT %MD936 : Real;   // Nhiệt độ giải nhiệt đích Bồn chứa 01
   AI_HMI_SP_Loc_Ap_Suat_Max AT %MD940 : Real;   // Ngưỡng áp suất cao trước màng lọc
   AI_HMI_SP_Time_Khuay_Bon1 AT %MD944 : Time;   // Thời gian khuấy Bồn 1
   AI_HMI_SP_Time_Khuay_Bon3 AT %MD948 : Time;   // Thời gian khuấy Bồn 3
   AI_HMI_SP_Time_Fwd AT %MD952 : Time;   // Thời gian khuấy chiều thuận
   AI_HMI_SP_Time_Rev AT %MD956 : Time;   // Thời gian khuấy chiều ngược
   AI_HMI_SP_Time_Sterilize AT %MD960 : Time;   // Thời gian giữ nhiệt thanh trùng
   AI_PLC1_Khuay_Bon1_Xong AT %M336.2 : Bool;   // Trạng thái tự động xong khuấy Bồn 1
   AI_PLC1_Khuay_Thuan_Bon2_Xong AT %M336.3 : Bool;   // Trạng thái tự động xong khuấy thuận Bồn 2
   AI_PLC1_Khuay_Nghich_Bon2_Xong AT %M336.4 : Bool;   // Trạng thái tự động xong khuấy ngược Bồn 2
   AI_PLC1_Thanh_Trung_Bon2_Xong AT %M336.5 : Bool;   // Trạng thái tự động xong thanh trùng Bồn 2
   AI_PLC2_Khuay_Bon3_Xong AT %M336.6 : Bool;   // Trạng thái tự động xong khuấy Bồn 3
   AI_PLC2_Khuay_Thuan_Bon4_Xong AT %M336.7 : Bool;   // Trạng thái tự động xong khuấy thuận Bồn 4
   AI_PLC2_Khuay_Nghich_Bon4_Xong AT %M337.0 : Bool;   // Trạng thái tự động xong khuấy ngược Bồn 4
   AI_PLC2_Thanh_Trung_Bon4_Xong AT %M337.1 : Bool;   // Trạng thái tự động xong thanh trùng Bồn 4
   AI_PLC1_Tip_Bon1_Auto_Done AT %M337.2 : Bool;   // Trạng thái tự động xong tip Bồn 1
   AI_PLC1_Tip_Bon2_Auto_Done AT %M337.3 : Bool;   // Trạng thái tự động xong tip Bồn 2
   AI_PLC2_Tip_Bon3_Auto_Done AT %M337.4 : Bool;   // Trạng thái tự động xong tip Bồn 3
   AI_PLC2_Tip_Bon4_Auto_Done AT %M337.5 : Bool;   // Trạng thái tự động xong tip Bồn 4
   AI_PLC1_Start_Edge_Old AT %M337.6 : Bool;   // Cờ nhớ cạnh lên nút Start PLC1
   AI_PLC1_Start_Edge_Edge AT %M337.7 : Bool;   // Xung cạnh lên nút Start PLC1
   AI_PLC2_Start_Edge_Old AT %M338.0 : Bool;   // Cờ nhớ cạnh lên nút Start PLC2
   AI_PLC2_Start_Edge_Edge AT %M338.1 : Bool;   // Xung cạnh lên nút Start PLC2
   AI_PID_Bon2_Enable AT %M338.2 : Bool;   // Cho phép PID Bồn 2
   AI_PID_Bon2_ManualEnable AT %M338.3 : Bool;   // Chế độ manual PID Bồn 2
   AI_PID_Bon2_Error AT %M338.4 : Bool;   // Lỗi khối PID Bồn 2
   AI_PID_Bon2_Reset_Eff AT %M338.5 : Bool;   // Reset hiệu dụng PID Bồn 2
   AI_PID_Bon4_Enable AT %M338.6 : Bool;   // Cho phép PID mô phỏng Bồn 4
   AI_PID_Bon4_ManualEnable AT %M338.7 : Bool;   // Chế độ manual PID Bồn 4
   AI_PID_Bon4_Error AT %M339.0 : Bool;   // Lỗi khối PID Bồn 4
   AI_PID_Bon4_Reset_Eff AT %M339.1 : Bool;   // Reset hiệu dụng PID Bồn 4
   AI_PID_Bon2_ErrorBits AT %MD964 : DWord;   // Mã lỗi DWORD PID Bồn 2
   AI_PID_Bon4_ErrorBits AT %MD968 : DWord;   // Mã lỗi DWORD PID Bồn 4
   AI_PID_Bon2_SP AT %MD972 : Real;   // Setpoint đưa vào PID Bồn 2
   AI_PID_Bon2_Err AT %MD976 : Real;   // Sai lệch PID Bồn 2 = SP - PV
   AI_PID_Bon2_CV AT %MD980 : Real;   // Giá trị điều khiển PID Bồn 2
   AI_PID_Bon2_ManualValue AT %MD984 : Real;   // Giá trị manual PID Bồn 2
   AI_PID_Bon4_SP AT %MD988 : Real;   // Setpoint đưa vào PID mô phỏng Bồn 4
   AI_PID_Bon4_Err AT %MD992 : Real;   // Sai lệch PID mô phỏng Bồn 4 = SP - PV
   AI_PID_Bon4_CV AT %MD996 : Real;   // Giá trị điều khiển PID mô phỏng Bồn 4
   AI_PID_Bon4_ManualValue AT %MD1000 : Real;   // Giá trị manual PID Bồn 4
   AI_TT3219_Bon4_Sim AT %MD1004 : Real;   // Nhiệt độ mô phỏng nội bộ cho PID Bồn 4
   AI_PID_Bon2_Temp_Inc AT %MD1008 : Real;   // Mức tăng nhiệt mô phỏng Bồn 2
   AI_PID_Bon4_Tang_Nhiet_Buoc AT %MD1012 : Real;   // Mức tăng nhiệt mô phỏng mỗi chu kỳ OB31
   AI_TT3219_Bon4_Target AT %MD1016 : Real;   // Nhiệt độ đích mô phỏng bồn 4
   AI_TT3219_Bon4_Sim_Pure AT %MD1020 : Real;   // Nhiệt độ mô phỏng chưa có nhiễu bồn 4
   AI_PID_Bon4_Temp_Val_1 AT %MD1024 : Real;   // Biến tạm mô phỏng nhiệt độ 1
   AI_PID_Bon4_Temp_Val_2 AT %MD1028 : Real;   // Biến tạm mô phỏng nhiệt độ 2
   AI_PID_Bon4_Sim_Counter AT %MD1032 : Real;   // Đồng hồ chu kỳ mô phỏng
   AI_PID_Bon4_Sim_Angle AT %MD1036 : Real;   // Góc lượng giác nhiễu
   AI_PID_Bon4_Sim_Sin AT %MD1040 : Real;   // Giá trị hình sin nhiễu
   AI_PID_Bon4_Sim_Noise AT %MD1044 : Real;   // Giá trị nhiễu nhiệt độ
   AI_PLC1_Tip_Bon1_Timer AT %MD1048 : Real;   // Bộ đếm thời gian mô phỏng tip bồn 1
   AI_PLC1_Tip_Bon2_Timer AT %MD1052 : Real;   // Bộ đếm thời gian mô phỏng tip bồn 2
   AI_PLC2_Tip_Bon3_Timer AT %MD1056 : Real;   // Bộ đếm thời gian mô phỏng tip bồn 3
   AI_PLC2_Tip_Bon4_Timer AT %MD1060 : Real;   // Bộ đếm thời gian mô phỏng tip bồn 4
   AI_PID_Bon2_State AT %MW534 : Int;   // Trạng thái khối PID Bồn 2
   AI_PLC1_Stop_Active AT %M339.2 : Bool;   // Tín hiệu dừng active PLC1
   AI_VFD_Bon2_Khuay_Active AT %M339.4 : Bool;   // Trạng thái khuấy Bồn 2 active
   AI_VFD_Bon2_Should_Run AT %M339.5 : Bool;   // Yêu cầu chạy VFD Bồn 2
   AI_HMI_Use_Sim_Input_PLC1 AT %M340.0 : Bool;   // Cho phép sử dụng đầu vào mô phỏng PLC1
   AI_HMI_Use_Sim_Input_BonChua AT %M340.2 : Bool;   // Cho phép sử dụng đầu vào mô phỏng Bồn chứa
   AI_PLC2_Me_Nhanh2_Hoan_Thanh_Nhan_Eff AT %M340.3 : Bool;   // Cờ nhận trạng thái hoàn thành Nhánh 2 hiệu dụng
   AI_PLC2_Me_Nhanh2_Hoan_Thanh_Nhan_HMI_Gated AT %M340.5 : Bool;   // Cờ nhận trạng thái hoàn thành Nhánh 2 HMI gated
   AI_PLC1_SP_Valid AT %M340.7 : Bool;   // Setpoint PLC1 hợp lệ
   AI_BonChua_SP_Valid AT %M341.1 : Bool;   // Setpoint Bồn chứa hợp lệ
   AI_PLC1_Loi_Setpoint AT %M341.2 : Bool;   // Lỗi Setpoint PLC1
   AI_BonChua_Loi_Setpoint AT %M341.4 : Bool;   // Lỗi Setpoint Bồn chứa
   AI_Init_Defaults_Done_PLC1 AT %M341.5 : Bool;   // Khởi tạo Setpoint mặc định PLC1 hoàn tất
   AI_Init_Defaults_Done_BonChua AT %M341.7 : Bool;   // Khởi tạo Setpoint mặc định Bồn chứa hoàn tất
   AI_Init_Trigger_PLC1 AT %M342.0 : Bool;   // Cờ kích hoạt nạp recipe mặc định PLC1
   AI_Init_Trigger_BonChua AT %M342.2 : Bool;   // Cờ kích hoạt nạp recipe mặc định Bồn chứa
   AI_HMI_Load_Default_Recipe AT %M342.3 : Bool;   // Yêu cầu nạp lại Recipe mặc định từ HMI
   AI_PLC1_Load_Default_Cmd AT %M342.4 : Bool;   // Lệnh nạp recipe mặc định gửi sang PLC2
   AI_PLC1_Load_Default_Cmd_M AT %M225.0 : Bool;   // Tag gương phản hồi HMI cho lệnh nạp recipe mặc định PLC1
   AI_PLC1_Load_Default_Done_Nhan AT %M343.1 : Bool;   // Nhận báo nạp recipe xong từ PLC2
   AI_PLC1_Load_Default_Done_Nhan_HMI AT %M111.7 : Bool;   // Tín hiệu mô phỏng/HMI cho nhận báo nạp recipe xong
   AI_PLC1_Load_Default_Done_Nhan_HMI_Gated AT %M343.2 : Bool;   // Tín hiệu nhận báo nạp recipe xong HMI gated
   AI_PLC1_Load_Default_Done_Nhan_Eff AT %M343.3 : Bool;   // Tín hiệu nhận báo nạp recipe xong hiệu dụng
   AI_HMI_Sim_Mode AT %M343.4 : Bool;   // Cho phép toàn bộ tín hiệu mô phỏng HMI tác động vào input hiệu dụng
   AI_HMI_Run_Enable AT %M343.5 : Bool;   // Cho phép vận hành từ HMI ở chế độ thật
   AI_System_Mode_Real AT %M343.6 : Bool;   // Hệ thống đang hoạt động ở chế độ thực tế
   AI_System_Mode_Sim AT %M343.7 : Bool;   // Hệ thống đang hoạt động ở chế độ mô phỏng
   AI_HMI_Sim_Active_Warning AT %M344.0 : Bool;   // Cảnh báo chế độ mô phỏng HMI đang hoạt động
   AI_PID_Bon2_Kp_HMI AT %MD1064 : Real;   // HMI parameter for Kp PID Bồn 2
   AI_PID_Bon2_Ti_HMI AT %MD1068 : Real;   // HMI parameter for Ti PID Bồn 2
   AI_BonChua_Nhan_Dich_Xong_Nhanh1 AT %M344.1 : Bool;   // Nhận dịch xong từ Nhánh 1
   AI_BonChua_Nhan_Dich_Xong_Nhanh2 AT %M344.2 : Bool;   // Nhận dịch xong từ Nhánh 2
   AI_Clock_1Hz_Last AT %M344.3 : Bool;   // Trạng thái Clock 1Hz chu kỳ trước
   AI_Clock_1Hz_Edge AT %M344.4 : Bool;   // Xung cạnh lên của Clock 1Hz
   AI_PLC2_Heartbeat_Last AT %MW540 : Int;   // Heartbeat PLC2 chu kỳ trước
   AI_PLC2_Heartbeat_Changed AT %M344.7 : Bool;   // Cờ heartbeat PLC2 thay đổi
   AI_PLC1_Heartbeat_Timeout AT %M345.0 : Bool;   // Lỗi timeout heartbeat PLC2
   AI_VFD_Bon2_MB_Req AT %M345.1 : Bool;   // REQ cho VFD Modbus
   AI_VFD_Bon2_MB_Mode AT %MB500 : USInt;   // MODE cho VFD Modbus
   AI_VFD_Bon2_MB_DataAddr AT %MD504 : UDInt;   // DATA_ADDR cho VFD Modbus
   AI_VFD_Bon2_MB_DataLen AT %MW508 : UInt;   // DATA_LEN cho VFD Modbus
   AI_VFD_Bon2_MB_DataBuffer AT %MW510 : Word;   // Buffer dữ liệu cho VFD Modbus
END_VAR

VAR_GLOBAL   // PLC tag table "All_Tags"
   CCC1 AT %I10.0 : Bool;
   CCC2 AT %I10.1 : Bool;
   Tag_1 AT %M5.6 : Bool;
   Tag_2 AT %M5.7 : Bool;
   Tag_3 AT %M6.0 : Bool;
   Tag_4 AT %M6.1 : Bool;
   Tag_5 AT %M6.2 : Bool;
   Tag_6 AT %M6.3 : Bool;
   Tag_7 AT %M6.4 : Bool;
   Tag_8 AT %M6.5 : Bool;
   Tag_9 AT %M6.6 : Bool;
END_VAR

VAR_GLOBAL   // PLC tag table "Assembly_tags"
   "Assembly green lid start" AT %I8.0 : Bool;
   "Assembly blue lid start" AT %I8.1 : Bool;
   "Assembly green base start" AT %I8.2 : Bool;
   "Assembly blue base start" AT %I8.3 : Bool;
   "G_lid in place" AT %I8.4 : Bool;
   "G_base in place" AT %I8.5 : Bool;
   G_lid_clamped AT %I8.6 : Bool;
   G_base_clamped AT %I8.7 : Bool;
   G_part_leaving AT %I9.0 : Bool;
   G_item_detect AT %I9.1 : Bool;
   "B_lid in place" AT %I9.2 : Bool;
   "B_base in place" AT %I9.3 : Bool;
   B_lid_clamped AT %I9.4 : Bool;
   B_base_clamped AT %I9.5 : Bool;
   B_part_leaving AT %I9.6 : Bool;
   B_item_detect AT %I9.7 : Bool;
   G_Negative_Trig_1 AT %M4.0 : Bool;
   G_Negative_Trig_2 AT %M4.1 : Bool;
   G_Negative_Trig_3 AT %M4.2 : Bool;
   move_green_lid_conv AT %M4.3 : Bool;
   move_green_base_conv AT %M4.4 : Bool;
   move_blue_lid_conv AT %M4.5 : Bool;
   move_blue_base_conv AT %M4.6 : Bool;
   B_Negative_Trig_1 AT %M4.7 : Bool;
   B_Negative_Trig_2 AT %M5.0 : Bool;
   B_Negative_Trig_3 AT %M5.1 : Bool;
   G_Detected_Memory AT %M5.2 : Bool;
   G_Reset AT %M5.3 : Bool;
   B_Detected_Memory AT %M5.4 : Bool;
   B_Reset AT %M5.5 : Bool;
   G_Timer_1 AT %T0 : Timer;
   G_Timer_2 AT %T1 : Timer;
   G_Timer_3 AT %T2 : Timer;
   B_Timer_1 AT %T3 : Timer;
   B_Timer_2 AT %T4 : Timer;
   B_Timer_3 AT %T5 : Timer;
   G_lids_conv_1 AT %Q7.0 : Bool;
   G_lids_conv_2 AT %Q7.1 : Bool;
   G_lids_conv_3 AT %Q7.2 : Bool;
   G_lids_conv_4 AT %Q7.3 : Bool;
   G_lids_conv_5 AT %Q7.4 : Bool;
   G_lids_conv_6 AT %Q7.5 : Bool;
   G_lids_conv_7 AT %Q7.6 : Bool;
   G_lids_conv_8 AT %Q7.7 : Bool;
   B_lids_conv_1 AT %Q8.0 : Bool;
   B_lids_conv_2 AT %Q8.1 : Bool;
   B_lids_conv_3 AT %Q8.2 : Bool;
   B_lids_conv_4 AT %Q8.3 : Bool;
   G_base_conv_1 AT %Q8.4 : Bool;
   G_base_conv_2 AT %Q8.5 : Bool;
   G_base_conv_3 AT %Q8.6 : Bool;
   G_base_conv_4 AT %Q8.7 : Bool;
   G_base_conv_5 AT %Q9.0 : Bool;
   G_base_conv_6 AT %Q9.1 : Bool;
   B_base_conv_1 AT %Q9.2 : Bool;
   B_base_conv_2 AT %Q9.3 : Bool;
   B_base_conv_3 AT %Q9.4 : Bool;
   B_base_conv_4 AT %Q9.5 : Bool;
   G_clamp_lid AT %Q9.6 : Bool;
   G_clamp_base AT %Q9.7 : Bool;
   "G_move Z" AT %Q10.0 : Bool;
   G_grab AT %Q10.1 : Bool;
   "G_move X" AT %Q10.2 : Bool;
   "G_pos.Raise_bases" AT %Q10.3 : Bool;
   B_clamp_lid AT %Q10.4 : Bool;
   B_clamp_base AT %Q10.5 : Bool;
   "B_move Z" AT %Q10.6 : Bool;
   B_grab AT %Q10.7 : Bool;
   "B_move X" AT %Q11.0 : Bool;
   "B_pos.Raise_bases" AT %Q11.1 : Bool;
END_VAR

VAR_GLOBAL   // PLC tag table "Default tag table"
   System_Byte AT %MB1 : Byte;
   FirstScan AT %M1.0 : Bool;
   DiagStatusUpdate AT %M1.1 : Bool;
   AlwaysTRUE AT %M1.2 : Bool;
   AlwaysFALSE AT %M1.3 : Bool;
   Clock_Byte AT %MB0 : Byte;
   Clock_10Hz AT %M0.0 : Bool;
   Clock_5Hz AT %M0.1 : Bool;
   "Clock_2.5Hz" AT %M0.2 : Bool;
   Clock_2Hz AT %M0.3 : Bool;
   "Clock_1.25Hz" AT %M0.4 : Bool;
   Clock_1Hz AT %M0.5 : Bool;
   "Clock_0.625Hz" AT %M0.6 : Bool;
   "Clock_0.5Hz" AT %M0.7 : Bool;
   PTRIG AT %M2.0 : Bool;
   PTRIG2 AT %M2.1 : Bool;
END_VAR

VAR_GLOBAL   // PLC tag table "INPUT"
   I_Mode AT %I0.0 : Bool;   // Switch chế độ 1 auto, 0 manu
   I_CB_Cao AT %I0.1 : Bool;   // Cảm biến sản phẩm cao
   I_CB_Trung_Binh AT %I0.2 : Bool;   // Cảm biến sản phẩm trung bình
   I_CB_Thap AT %I0.3 : Bool;   // Cảm biến sản phẩm thấp
   I_BT AT %I0.4 : Bool;   // Chạy/Dừng động cơ băng tải
   I_Xylanh_Cao AT %I0.5 : Bool;   // Đóng/mở xi lanh sản phẩm cao
   I_Xylanh_TB AT %I0.6 : Bool;   // Đóng/mở xi lanh sản phẩm trung bình
END_VAR

VAR_GLOBAL   // PLC tag table "INPUT_M"
   M_Mode AT %M10.0 : Bool;   // Switch chế độ 1 auto, 0 manu
   M_CB_Cao AT %M10.1 : Bool;   // Cảm biến sản phẩm cao
   M_CB_Trung_Binh AT %M10.2 : Bool;   // Cảm biến sản phẩm trung bình
   M_CB_Thap AT %M10.3 : Bool;   // Cảm biến sản phẩm thấp
   M_BT AT %M10.4 : Bool;   // Chạy/Dừng động cơ băng tải
   M_Xylanh_Cao AT %M10.5 : Bool;   // Đóng/mở xi lanh sản phẩm cao
   M_Xylanh_TB AT %M10.6 : Bool;   // Đóng/mở xi lanh sản phẩm trung bình
END_VAR

VAR_GLOBAL   // PLC tag table "OUTPUT"
   Q_lamp_Auto AT %Q0.0 : Bool;   // Đèn chế độ auto
   Q_lamp_Manu AT %Q0.1 : Bool;   // Đèn chế độ manu
   Q_BT AT %Q0.2 : Bool;   // Băng tải phân loại
   Q_Xylanh_Cao AT %Q0.3 : Bool;   // Xi lanh đẩy sản phẩm cao
   Q_Xylanh_TB AT %Q0.4 : Bool;   // Xi lanh đẩy sản phẩm trung bình
END_VAR

VAR_GLOBAL   // PLC tag table "PTRIG"
   P1 AT %M330.0 : Bool;
   P2 AT %M330.1 : Bool;
   P3 AT %M330.2 : Bool;
   P4 AT %M330.3 : Bool;
   P5 AT %M330.4 : Bool;
   P6 AT %M330.5 : Bool;
   P7 AT %M330.6 : Bool;
   P8 AT %M330.7 : Bool;
   P9 AT %M331.0 : Bool;
   P10 AT %M331.1 : Bool;
   P11 AT %M331.2 : Bool;
END_VAR

VAR_GLOBAL   // PLC tag table "SO_NGUYEN"
   Act_Count_Cao AT %MW200 : Int;   // Bộ đếm số sản phẩm trọng lượng nhẹ
   Act_Count_TB AT %MW202 : Int;   // Bộ đếm số sản phẩm trọng lượng trung bình
   Act_Count_Thap AT %MW204 : Int;   // Bộ đếm số sản phẩm trọng lượng nặng
   Simu_VT_SP AT %MW206 : Int;   // Mô phỏng vị trí sản phẩm
   Simu_Type_SP AT %MW208 : Int;   // Mô phỏng loại sản phẩm
END_VAR

VAR_GLOBAL   // PLC tag table "TAG"
   Start AT %I0.0 : Bool;   // Nút nhấn Start
   Stop AT %I0.1 : Bool;   // Nút nhấn Stop
   Lamp AT %Q0.0 : Bool;   // Đèn hệ thống làm việc
   Sensor_Temperature AT %IW64 : Int;   // Cảm biến nhiệt độ
   QW_SSR AT %QW64 : Int;   // Đầu ra analog điều khiển SSR
   HMI_Start AT %M10.0 : Bool;   // Nút nhấn start trên Scada
   HMI_Stop AT %M10.1 : Bool;   // Nút nhấn Stop trên Scada
   HMI_Simulation AT %M10.2 : Bool;   // Nút mô phỏng tín hiệu nhiệt độ trên Scada
   HMI_Simu_Temperature AT %MW100 : Int;   // Mô phỏng nhiệt độ trên HMI
   HMI_Setting_Temperature AT %MD200 : Real;   // Cài đặt nhiệt độ cho máy sấy
   HMI_TT_Temperature AT %MD204 : Real;   // Nhiệt độ thực tế máy sấy
END_VAR

VAR_GLOBAL   // PLC tag table "TRUNGGIAN"
   Q_Auto_BT AT %M20.0 : Bool;   // Băng tải phân loại
   Q_Auto_Xylanh_Cao AT %M20.1 : Bool;   // Xi lanh đẩy sản phẩm cao
   Q_Auto_Xylanh_TB AT %M20.2 : Bool;   // Xi lanh đẩy sản phẩm trung bình
   Q_Manu_BT AT %M30.0 : Bool;   // Băng tải phân loại
   Q_Manu_Xylanh_Cao AT %M30.1 : Bool;   // Xi lanh đẩy sản phẩm cao
   Q_Manu_Xylanh_TB AT %M30.2 : Bool;   // Xi lanh đẩy sản phẩm trung bình
   M_Simulation AT %M5.0 : Bool;   // Nút mô phỏng trên scada
   M_Reset AT %M5.1 : Bool;   // Nút reset
   SIMU_CB_CAO AT %M5.2 : Bool;   // Mô phỏng cảm biến cao
   SIMU_CB_TB AT %M5.3 : Bool;   // Mô phỏng cảm biến trung bình
   SIMU_CB_THAP AT %M5.4 : Bool;   // Mô phỏng cảm biến thấp
END_VAR

VAR_GLOBAL   // PLC tag table "base_feeding_station"
   lid_detection AT %I0.0 : Bool;
   stop_beginning_lid_sensor AT %I0.1 : Bool;
   start_LID_feeding_convyer AT %I0.2 : Bool;
   LID_detected_grip AT %I0.3 : Bool;
   stop_LID_Feeding AT %I0.4 : Bool;
   LID_machining_entrance_sensor AT %I0.5 : Bool;
   base_Raw_counter_start AT %I0.6 : Bool;
   stop_base_begininning_convyr AT %I0.7 : Bool;
   base_gripper_detected AT %I1.0 : Bool;
   start_base_raw_feeding AT %I1.1 : Bool;
   stop_base_raw_feeding AT %I1.2 : Bool;
   stop_base_machining_convyr AT %I1.3 : Bool;
   lid_start_button AT %I1.4 : Bool;
   lid_stop_button AT %I1.5 : Bool;
   lid_emergency_button AT %I1.6 : Bool;
   base_start_button AT %I1.7 : Bool;
   base_stop_button AT %I2.0 : Bool;
   base_emergency AT %I2.1 : Bool;
   Lid_beginning_conveyr AT %Q0.0 : Bool;
   lid_feeding_conveyr AT %Q0.1 : Bool;
   Lid_pickup_x_axis AT %Q0.3 : Bool;
   lid_pickup_z_axis AT %Q0.4 : Bool;
   lid_sucction_gripper AT %Q0.5 : Bool;
   base_beginning_conveyr AT %Q0.6 : Bool;
   "lid-machinning_conveyr" AT %Q0.2 : Bool;
   base_raw_feeding_conveyr AT %Q0.7 : Bool;
   base_to_machinning_conveyr AT %Q1.0 : Bool;
   base_pickup_x_axis AT %Q1.1 : Bool;
   base_pickup_z_axis AT %Q1.2 : Bool;
   base_sucction_gripper AT %Q1.3 : Bool;
   base_start_button_1_light AT %Q1.4 : Bool;
   base_stop_button_1_light AT %Q1.5 : Bool;
   lid_start_light AT %Q1.6 : Bool;
   lid_stop_button_1_light AT %Q1.7 : Bool;
   base_raw_material AT %Q2.0 : Bool;
   lid_raw_emit AT %Q2.1 : Bool;
   state_of_start_base AT %M0.0 : Bool;
   state_of_start_LID AT %M0.1 : Bool;
   state_of_lid AT %M0.2 : Bool;
   dummy AT %M0.3 : Bool;
   To_emit_lid AT %M0.4 : Bool;
   item_ready_to_picked AT %M0.5 : Bool;
   movin_lid_z_mem AT %M0.6 : Bool;
   LID_moving_z_sensor AT %I2.4 : Bool;
   LID_moving_x_sensor AT %I2.5 : Bool;
   "dummy(1)" AT %M0.7 : Bool;
   "dummy(2)" AT %M1.0 : Bool;
   lid_belt_convyer_excess AT %Q2.2 : Bool;
   push_excess_blue_lid AT %Q2.3 : Bool;
   push_excess_green_lid AT %Q2.4 : Bool;
   Blue_vision_lid AT %I2.6 : Bool;
   green_vision_lid AT %I2.7 : Bool;
   front_blue_push_lid AT %I3.0 : Bool;
   back_blue_push_lid AT %I3.1 : Bool;
   front_green_push_lid AT %I3.2 : Bool;
   back_green_push_lid AT %I3.3 : Bool;
   into_cnc_lid_sensor AT %I3.4 : Bool;
   CNC_lid_empty AT %M1.1 : Bool;
   ONE_OBJECT_IN AT %Q2.5 : Bool;
   KEEP_DISTANCE AT %Q2.6 : Bool;
   ARE_WE_THERE_YET_BLUE_lid AT %M1.2 : Bool;
   ARE_WE_THERE_YET_GREEN_lid AT %M1.3 : Bool;
   LID_COUNTER_RESET_BUTTON_BLUE AT %I3.5 : Bool;
   TO_STORAGE_BLUE_CONVYER_lid AT %Q2.7 : Bool;
   TO_STORAGE_GREEN_CONVYER_lid AT %Q3.0 : Bool;
   TO_STORAGE_BLUE_SENSOR_lid AT %I3.6 : Bool;
   TO_STORAGE_GREEN_SENSOR_lid AT %I3.7 : Bool;
   LID_COUNTER_RESET_BUTTON_GREEN AT %I4.0 : Bool;
   "GREEN_LID_PUSHER_SORTING(FRONT LIMIT)" AT %I4.1 : Bool;
   "GREEN_LID_PUSHER_SORTING(BACK LIMITT)" AT %I4.2 : Bool;
   "BLUE_LID_PUSHER_SORTING(FRONT LIMIT)" AT %I4.3 : Bool;
   "BLUE_LID_PUSHER_SORTING(BACK LIMIT)" AT %I4.4 : Bool;
   BEGIN_SORTING_STATION_LIDS AT %I4.5 : Bool;
   BLUE_LID_VISION_SORTING AT %I4.6 : Bool;
   GREEN_LID_VISION_SORTING AT %I4.7 : Bool;
   SORTING_CONVYER_LID AT %Q3.1 : Bool;
   GREEN_LID_PUSHER_SORTING AT %Q3.2 : Bool;
   BLUE_LID_PUSHER_SORTING AT %Q3.3 : Bool;
   CNC_base_empty AT %M2.5 : Bool;
   to_emit_base AT %M1.5 : Bool;
   base_into_cnc AT %I5.0 : Bool;
   BASE_MOVE_X_SENSOR AT %I5.1 : Bool;
   BASE_MOVE_Z_SENSOR AT %I5.2 : Bool;
   DUMMY1 AT %M1.6 : Bool;
   DUMMY2 AT %M1.7 : Bool;
   DUMMY3 AT %M2.0 : Bool;
   DUMMY4 AT %M2.1 : Bool;
   DUMMY5 AT %M2.2 : Bool;
   BASE_RAW_EXESS_CONV AT %Q3.4 : Bool;
   Are_we_there_base_raw_blue AT %M2.3 : Bool;
   Are_we_there_base_raw_green AT %M2.4 : Bool;
   base_raw_blue_exes_vision AT %I5.3 : Bool;
   base_raw_green_exes_vision AT %I5.4 : Bool;
   to_blue_base_raw_storage_sensor AT %I5.5 : Bool;
   to_green_base_raw_storage_sensor AT %I5.6 : Bool;
   "push_ex_green_base raw(front)" AT %I5.7 : Bool;
   "push_ex_green_base raw (back)" AT %I6.0 : Bool;
   "pusher blue base raw (front)" AT %I6.1 : Bool;
   "pusher blue base raw (back)" AT %I6.2 : Bool;
   is_base_exsist AT %M1.4 : Bool;
   Conv_sorting_set_base AT %M2.6 : Bool;
   BEGIN_SORTING_STATION_BASE_4 AT %Q5.3 : Bool;
END_VAR

VAR_GLOBAL   // PLC tag table "PLC1_Tags"
   Start_Cmd AT %M0.0 : Bool;
   Stop_Cmd AT %M0.1 : Bool;
   bMotorRunning AT %M0.2 : Bool;
   Reset_Cmd AT %M0.3 : Bool;
   DIR_Cmd AT %M0.4 : Bool;
   PID_Setpoint AT %MD10 : Real;
   PID_ProcessValue AT %MD14 : Real;
   PID_Output AT %MD18 : Real;
   Speed_SP_toSend AT %MD22 : Real;
   Speed_PV_from2 AT %MD26 : Real;
   ATV12_Status AT %MW30 : Word;
   Control_Byte AT %MB32 : Byte;
   Clock_1Hz AT %M100.5 : Bool;
   GET_NDR AT %M1.0 : Bool;
   GET_Error AT %M1.1 : Bool;
   GET_Status AT %MW2 : Word;
   PUT_NDR AT %M1.2 : Bool;
   PUT_Error AT %M1.3 : Bool;
   PUT_Status AT %MW4 : Word;
END_VAR

VAR_GLOBAL   // PLC tag table "Encoder_Tags"
   HSC_1_Value AT %ID1000 : DInt;   // Giá trị đếm xung thời kỳ thực từ bộ đếm tốc độ cao HSC1   {ExternalWritable false}
END_VAR

VAR_GLOBAL   // PLC tag table "PLC2_Tags"
   MB_ControlWord AT %MW40 : Word;
   MB_FreqSetpoint AT %MW42 : Int;
   MB_StatusWord AT %MW44 : Word;
   MB_ActualSpeed AT %MW46 : Int;
   MB_Error AT %M50.0 : Bool;
   MB_Busy AT %M50.1 : Bool;
   MB_Done AT %M50.2 : Bool;
   MB_Status AT %MW52 : Word;
   iStep AT %MW60 : Int;
   Freq_Temp AT %MD70 : Real;
   Speed_Actual_Temp AT %MD74 : Real;
   FirstScan AT %M101.0 : Bool;
   Clock_1Hz AT %M100.5 : Bool;
   MBCL_Done AT %M51.0 : Bool;
   MBCL_Error AT %M51.1 : Bool;
   MBCL_Status AT %MW54 : Word;
END_VAR

VAR_GLOBAL   // PLC tag table "Standard-Variablentabelle"
   start AT %I0.0 : Bool;
   stop AT %I0.1 : Bool;
   drain AT %I0.2 : Bool;
   levelMeter AT %ID30 : Real;
   SetPoint AT %ID38 : Real;
   FillValve AT %QD30 : Real;
   DissValve AT %QD34 : Real;
   SetPointDisplay AT %QD38 : DInt;
   LevelDisplay AT %QD42 : DInt;
   ErrorDisplay AT %QD46 : Real;
   Tag_1 AT %M0.0 : Bool;
   Tag_2 AT %MD100 : Real;
   scaledlevel AT %MW2 : Int;
   setscaled AT %MW12 : Int;
   Tag_3 AT %M2.2 : Bool;
END_VAR

DATA_BLOCK "AI_Timers_PLC1"   // DB
TITLE = AI_Timers_PLC1
{ S7_Optimized_Access := 'TRUE' }
VERSION : 0.1
// Global DB containing all timers and PID instances
// stored: AutoNumber true, IsOnlyStoredInLoadMemory false, IsWriteProtectedInAS false
   VAR
      AI_Timer_Dosing_Bon1 : IEC_TIMER;
      AI_Timer_Tip_Bon1 : IEC_TIMER;
      AI_Timer_Dosing_Bon2 : IEC_TIMER;
      AI_Timer_Tip_Bon2 : IEC_TIMER;
      AI_Timer_Khuay_Bon1 : IEC_TIMER;
      AI_Timer_Khuay_Thuan_Bon2 : IEC_TIMER;
      AI_Timer_Khuay_Nghich_Bon2 : IEC_TIMER;
      AI_Timer_Thanh_Trung_Bon2 : IEC_TIMER;
      AI_Timer_DryRun_Bon2 : IEC_TIMER;
      AI_Timer_Heartbeat_PLC1 : IEC_TIMER;
      AI_VFD_Bon2_MB_Counter : IEC_COUNTER;
   END_VAR
BEGIN
END_DATA_BLOCK

DATA_BLOCK "DB_PLC1_MB_Buffer_DB"   // DB12
TITLE = DB_PLC1_MB_Buffer_DB
{ S7_Optimized_Access := 'FALSE' }
VERSION : 0.1
// DB communication via Modbus TCP
// stored: AutoNumber false, IsOnlyStoredInLoadMemory false, IsWriteProtectedInAS false
   VAR
      Send_CmdSeq : Int;
      Send_Cmd_Start : Bool;
      Send_Cmd_Stop : Bool;
      Send_Cmd_Reset : Bool;
      Send_Cmd_EStop : Bool;
      Send_Cmd_Pump_Branch2_To_SubTanks : Bool;
      Send_Cmd_Load_Recipe : Bool;
      Send_Heartbeat : Int;
      Recv_AckSeq : Int;
      Recv_Done_Branch2 : Bool;
      Recv_Done_Recipe : Bool;
      Recv_Alarm : Bool;
      Recv_State : Int;
      Recv_PID_Bon4_SP : Real;
      Recv_PID_Bon4_PV : Real;
      Recv_PID_Bon4_CV : Real;
      Recv_Done_Discharge2 : Bool;
      Recv_Heartbeat : Int;
   END_VAR
BEGIN
END_DATA_BLOCK

DATA_BLOCK "DB_PLC1_Recv_From_PLC2_DB"   // DB10
TITLE = DB_PLC1_Recv_From_PLC2_DB
{ S7_Optimized_Access := 'FALSE' }
VERSION : 0.1
// DB communication via Modbus TCP
// stored: AutoNumber false, IsOnlyStoredInLoadMemory false, IsWriteProtectedInAS false
   VAR
      AckSeq : Int;
      Done_Branch2 : Bool;
      Done_Recipe : Bool;
      Alarm : Bool;
      State : Int;
      PID_Bon4_SP : Real;
      PID_Bon4_PV : Real;
      PID_Bon4_CV : Real;
      Done_Discharge2 : Bool;
      Heartbeat : Int;
   END_VAR
BEGIN
END_DATA_BLOCK

DATA_BLOCK "DB_PLC1_Send_To_PLC2_DB"   // DB11
TITLE = DB_PLC1_Send_To_PLC2_DB
{ S7_Optimized_Access := 'FALSE' }
VERSION : 0.1
// DB communication via Modbus TCP
// stored: AutoNumber false, IsOnlyStoredInLoadMemory false, IsWriteProtectedInAS false
   VAR
      CmdSeq : Int;
      Cmd_Start : Bool;
      Cmd_Stop : Bool;
      Cmd_Reset : Bool;
      Cmd_EStop : Bool;
      Cmd_Pump_Branch2_To_SubTanks : Bool;
      Cmd_Load_Recipe : Bool;
      Heartbeat : Int;
   END_VAR
BEGIN
END_DATA_BLOCK

DATA_BLOCK "AI_Timers_PLC2"   // DB
TITLE = AI_Timers_PLC2
{ S7_Optimized_Access := 'TRUE' }
VERSION : 0.1
// Global DB containing all timers and PID instances
// stored: AutoNumber true, IsOnlyStoredInLoadMemory false, IsWriteProtectedInAS false
   VAR
      AI_Timer_Dosing_Bon3 : IEC_TIMER;
      AI_Timer_Tip_Bon3 : IEC_TIMER;
      AI_Timer_Dosing_Bon4 : IEC_TIMER;
      AI_Timer_Tip_Bon4 : IEC_TIMER;
      AI_Timer_Khuay_Bon3 : IEC_TIMER;
      AI_Timer_Khuay_Thuan_Bon4 : IEC_TIMER;
      AI_Timer_Khuay_Nghich_Bon4 : IEC_TIMER;
      AI_Timer_Thanh_Trung_Bon4 : IEC_TIMER;
      AI_Timer_DryRun_Bon4 : IEC_TIMER;
      AI_Timer_Heartbeat_PLC2 : IEC_TIMER;
   END_VAR
BEGIN
END_DATA_BLOCK

DATA_BLOCK "DB_Modbus_Holding_Register_DB"   // DB20
TITLE = DB_Modbus_Holding_Register_DB
{ S7_Optimized_Access := 'FALSE' }
VERSION : 0.1
// DB communication via Modbus TCP
// stored: AutoNumber false, IsOnlyStoredInLoadMemory false, IsWriteProtectedInAS false
   VAR
      CmdSeq : Int;
      Cmd_Start : Bool;
      Cmd_Stop : Bool;
      Cmd_Reset : Bool;
      Cmd_EStop : Bool;
      Cmd_Pump_Branch2_To_SubTanks : Bool;
      Cmd_Load_Recipe : Bool;
      Heartbeat_Client : Int;
      AckSeq : Int;
      Done_Branch2 : Bool;
      Done_Recipe : Bool;
      Alarm : Bool;
      State : Int;
      PID_Bon4_SP : Real;
      PID_Bon4_PV : Real;
      PID_Bon4_CV : Real;
      Done_Discharge2 : Bool;
      Heartbeat_Server : Int;
   END_VAR
BEGIN
END_DATA_BLOCK

DATA_BLOCK "DB_MB_Client_Conn"   // DB11
TITLE = DB_MB_Client_Conn
{ S7_Optimized_Access := 'FALSE' }
VERSION : 0.1
// DB communication via Modbus TCP
// stored: AutoNumber false, IsOnlyStoredInLoadMemory false, IsWriteProtectedInAS false
   VAR
      MB_TCP : TCON_IP_v4;
   END_VAR
BEGIN
END_DATA_BLOCK

DATA_BLOCK "DB_MB_Client_Data"   // DB10
TITLE = DB_MB_Client_Data
{ S7_Optimized_Access := 'FALSE' }
VERSION : 0.1
// DB communication via Modbus TCP
// stored: AutoNumber false, IsOnlyStoredInLoadMemory false, IsWriteProtectedInAS false
   VAR
      Send_Words : Array[0..2] of Int;
      Recv_Words : Array[0..9] of Int;
   END_VAR
BEGIN
END_DATA_BLOCK

DATA_BLOCK "DB_MB_Server_Conn"   // DB13
TITLE = DB_MB_Server_Conn
{ S7_Optimized_Access := 'FALSE' }
VERSION : 0.1
// DB communication via Modbus TCP
// stored: AutoNumber false, DBAccessibleFromOPCUA true, IsOnlyStoredInLoadMemory false, IsWriteProtectedInAS false
   VAR
      MB_TCP_SERVER : TCON_IP_v4;
   END_VAR
BEGIN
END_DATA_BLOCK

DATA_BLOCK "DB_Modbus_Holding_Register"   // DB12
TITLE = DB_Modbus_Holding_Register
{ S7_Optimized_Access := 'FALSE' }
VERSION : 0.1
// DB communication via Modbus TCP
// stored: AutoNumber false, DBAccessibleFromOPCUA true, IsOnlyStoredInLoadMemory false, IsWriteProtectedInAS false
   VAR
      CmdSeq : Int;
      CmdBools : Int;
      Heartbeat_Client : Int;
      AckSeq : Int;
      StatusBools : Int;
      State : Int;
      PID_Bon4_SP : Real;
      PID_Bon4_PV : Real;
      PID_Bon4_CV : Real;
      Heartbeat_Server : Int;
   END_VAR
BEGIN
END_DATA_BLOCK

DATA_BLOCK "DB_MB_TCP_Client_Conn_DB"   // DB15
TITLE = DB_MB_TCP_Client_Conn_DB
{ S7_Optimized_Access := 'FALSE' }
VERSION : 0.1
// DB communication via Modbus TCP
// stored: AutoNumber false, DBAccessibleFromOPCUA true, IsOnlyStoredInLoadMemory false, IsWriteProtectedInAS false
   VAR
      MB_TCP : TCON_IP_v4;
   END_VAR
BEGIN
END_DATA_BLOCK

DATA_BLOCK "DB_MB_TCP_Server_Conn_DB"   // DB16
TITLE = DB_MB_TCP_Server_Conn_DB
{ S7_Optimized_Access := 'FALSE' }
VERSION : 0.1
// DB communication via Modbus TCP
// stored: AutoNumber false, DBAccessibleFromOPCUA true, IsOnlyStoredInLoadMemory false, IsWriteProtectedInAS false
   VAR
      MB_TCP_SERVER : TCON_IP_v4;
   END_VAR
BEGIN
END_DATA_BLOCK

DATA_BLOCK "DB10_NhanTuPLC2"   // DB10
{ S7_Optimized_Access := 'FALSE' }
VERSION : 0.1
// stored: AutoNumber true, IsOnlyStoredInLoadMemory false, IsWriteProtectedInAS false
   VAR
      Speed_Actual_fromPLC2 : Real;
      ATV12_Status_fromPLC2 : Word;
   END_VAR
BEGIN
END_DATA_BLOCK

DATA_BLOCK "DB11_GuiSangPLC2"   // DB11
{ S7_Optimized_Access := 'FALSE' }
VERSION : 0.1
// stored: AutoNumber true, IsOnlyStoredInLoadMemory false, IsWriteProtectedInAS false
   VAR
      Speed_SP_toSend : Real;
      Control_Byte_toSend : Bool;
      Reset_Cmd_toSend : Bool;
      DIR_Cmd_toSend : Bool;
   END_VAR
BEGIN
END_DATA_BLOCK

DATA_BLOCK "DB1_NhanTuPLC1"   // DB1
{ S7_Optimized_Access := 'FALSE' }
VERSION : 0.1
// stored: AutoNumber true, IsOnlyStoredInLoadMemory false, IsWriteProtectedInAS false
   VAR
      Speed_SP_fromPLC1 : Real;
      Control_Byte : Bool;
      Reset_Cmd : Bool;
      DIR_Cmd : Bool;
   END_VAR
BEGIN
END_DATA_BLOCK

DATA_BLOCK "DB2_GuiVePLC1"   // DB2
{ S7_Optimized_Access := 'FALSE' }
VERSION : 0.1
// stored: AutoNumber true, IsOnlyStoredInLoadMemory false, IsWriteProtectedInAS false
   VAR
      Speed_Actual_toSend : Real;
      ATV12_Status_toSend : Word;
   END_VAR
BEGIN
END_DATA_BLOCK

DATA_BLOCK "DB3_Encoder"   // DB5
TITLE = Encoder HSC Data Block
{ S7_Optimized_Access := 'FALSE' }
VERSION : 0.1
// Khối dữ liệu chứa tham số và trạng thái Encoder HSC1
// stored: AutoNumber true, IsOnlyStoredInLoadMemory false, IsWriteProtectedInAS false
   VAR
      Encoder_Count_Current : DInt;
      Encoder_Count_Last : DInt;
      Encoder_Count_Delta : DInt;
      Encoder_Count_Delta_Real : Real;
      Encoder_PPR : Real := 1000.0;
      Encoder_Effective_PPR : Real;
      Encoder_SampleTime_s : Real := 0.1;
      Encoder_RPM : Real;
      Encoder_Hz_Raw : Real;
      Encoder_Hz : Real;
      Encoder_Feedback_Selected : Real;
      Encoder_Use_Feedback : Bool := true;
      Encoder_Fault : Bool;
      Encoder_Use_Fourfold : Bool := true;
      Encoder_Motor_Pole_Pairs : Real := 2.0;
      Encoder_Fallback_Active : Bool;
      Encoder_NoPulse_Count : Real;
      Encoder_NoPulse_Limit : Real := 30.0;
   END_VAR
BEGIN
END_DATA_BLOCK

DATA_BLOCK "hmi"   // DB5
{ S7_Optimized_Access := 'TRUE' }
VERSION : 0.1
// stored: AutoNumber true, IsOnlyStoredInLoadMemory false, IsRetainMemResEnabled false, IsWriteProtectedInAS false, MemoryReserve 100
   VAR
      startfromhmi : Bool;
   END_VAR
BEGIN
END_DATA_BLOCK

ORGANIZATION_BLOCK "Main"   // OB1, LAD, ProgramCycle
TITLE = "Main Program Sweep (Cycle)"
{ S7_Optimized_Access := 'TRUE' }
VERSION : 0.1
// stored: AutoNumber true, IsIECCheckEnabled false, SetENOAutomatically false
   VAR_INPUT
      Initial_Call : Bool;   // Initial call of this OB
      Remanence : Bool;   // =True, if remanent data are available
   END_VAR
BEGIN

REGION Network 1
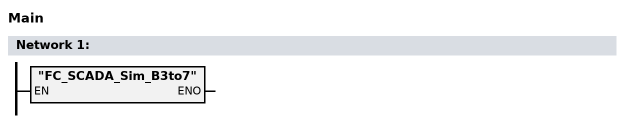
   RUNG wire#powerrail
      "FC_SCADA_Sim_B3to7"()
   END_RUNG
   // the same network as SCL:
   "FC_SCADA_Sim_B3to7"();
END_REGION
END_ORGANIZATION_BLOCK

ORGANIZATION_BLOCK "OB30_PID_PLC1_Bon2"   // OB30, LAD, CyclicInterrupt
{ S7_Optimized_Access := 'TRUE' }
VERSION : 0.1
// stored: AutoNumber true, IsIECCheckEnabled false
   VAR_INPUT
      Initial_Call : Bool;
      Remanence : Bool;
   END_VAR
BEGIN

REGION Network 1: Initialize PID Bon 2 Kp parameter
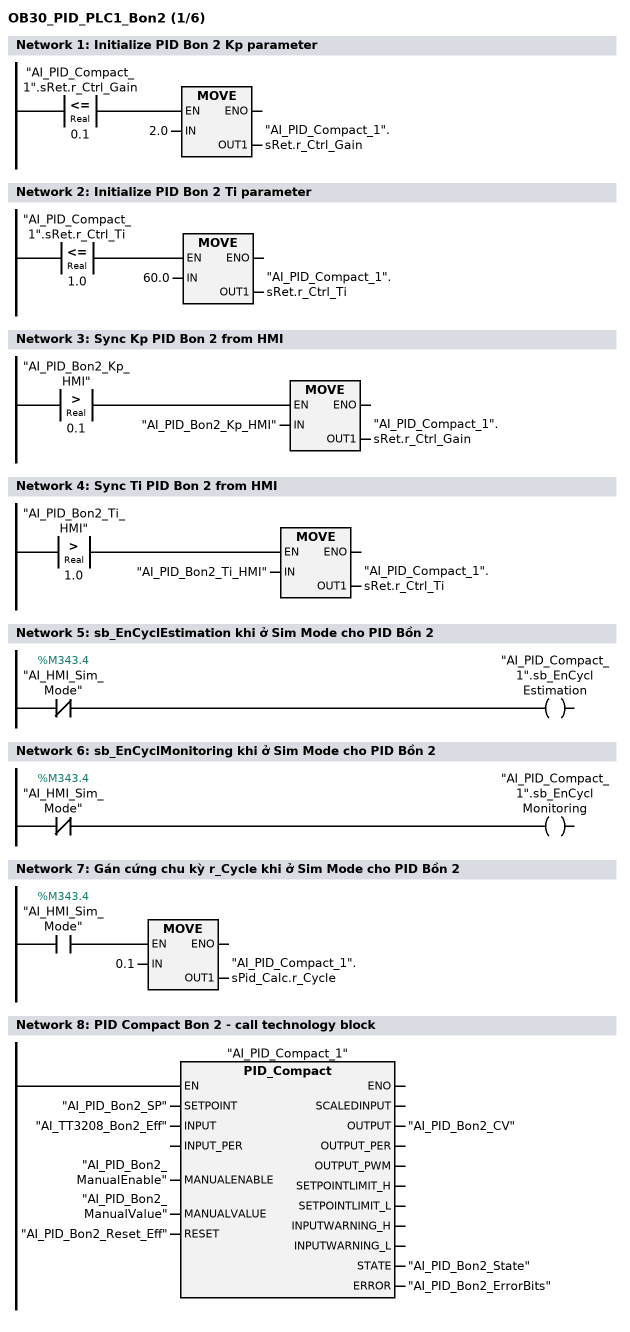
   RUNG wire#powerrail
      { S7_Templates := "SrcType := Real" } LE_Contact(in1 := "AI_PID_Compact_1".sRet.r_Ctrl_Gain, in2 := 0.1)
      { S7_GenerateENO := "TRUE" } Move(in := 2.0, out1 => "AI_PID_Compact_1".sRet.r_Ctrl_Gain)
   END_RUNG
   // the same network as SCL:
   IF "AI_PID_Compact_1".sRet.r_Ctrl_Gain <= 0.1 THEN "AI_PID_Compact_1".sRet.r_Ctrl_Gain := 2.0; END_IF;
END_REGION

REGION Network 2: Initialize PID Bon 2 Ti parameter
   RUNG wire#powerrail
      { S7_Templates := "SrcType := Real" } LE_Contact(in1 := "AI_PID_Compact_1".sRet.r_Ctrl_Ti, in2 := 1.0)
      { S7_GenerateENO := "TRUE" } Move(in := 60.0, out1 => "AI_PID_Compact_1".sRet.r_Ctrl_Ti)
   END_RUNG
   // the same network as SCL:
   IF "AI_PID_Compact_1".sRet.r_Ctrl_Ti <= 1.0 THEN "AI_PID_Compact_1".sRet.r_Ctrl_Ti := 60.0; END_IF;
END_REGION

REGION Network 3: Sync Kp PID Bon 2 from HMI
   RUNG wire#powerrail
      { S7_Templates := "SrcType := Real" } GT_Contact(in1 := "AI_PID_Bon2_Kp_HMI", in2 := 0.1)
      { S7_GenerateENO := "TRUE" } Move(in := "AI_PID_Bon2_Kp_HMI", out1 => "AI_PID_Compact_1".sRet.r_Ctrl_Gain)
   END_RUNG
   // the same network as SCL:
   IF "AI_PID_Bon2_Kp_HMI" > 0.1 THEN "AI_PID_Compact_1".sRet.r_Ctrl_Gain := "AI_PID_Bon2_Kp_HMI"; END_IF;
END_REGION

REGION Network 4: Sync Ti PID Bon 2 from HMI
   RUNG wire#powerrail
      { S7_Templates := "SrcType := Real" } GT_Contact(in1 := "AI_PID_Bon2_Ti_HMI", in2 := 1.0)
      { S7_GenerateENO := "TRUE" } Move(in := "AI_PID_Bon2_Ti_HMI", out1 => "AI_PID_Compact_1".sRet.r_Ctrl_Ti)
   END_RUNG
   // the same network as SCL:
   IF "AI_PID_Bon2_Ti_HMI" > 1.0 THEN "AI_PID_Compact_1".sRet.r_Ctrl_Ti := "AI_PID_Bon2_Ti_HMI"; END_IF;
END_REGION

REGION Network 5: sb_EnCyclEstimation khi ở Sim Mode cho PID Bồn 2
   RUNG wire#powerrail
      I_Contact( "AI_HMI_Sim_Mode" )
      Coil( "AI_PID_Compact_1".sb_EnCyclEstimation )
   END_RUNG
   // the same network as SCL:
   "AI_PID_Compact_1".sb_EnCyclEstimation := NOT "AI_HMI_Sim_Mode";
END_REGION

REGION Network 6: sb_EnCyclMonitoring khi ở Sim Mode cho PID Bồn 2
   RUNG wire#powerrail
      I_Contact( "AI_HMI_Sim_Mode" )
      Coil( "AI_PID_Compact_1".sb_EnCyclMonitoring )
   END_RUNG
   // the same network as SCL:
   "AI_PID_Compact_1".sb_EnCyclMonitoring := NOT "AI_HMI_Sim_Mode";
END_REGION

REGION Network 7: Gán cứng chu kỳ r_Cycle khi ở Sim Mode cho PID Bồn 2
   RUNG wire#powerrail
      Contact( "AI_HMI_Sim_Mode" )
      { S7_GenerateENO := "TRUE" } Move(in := 0.1, out1 => "AI_PID_Compact_1".sPid_Calc.r_Cycle)
   END_RUNG
   // the same network as SCL:
   IF "AI_HMI_Sim_Mode" THEN "AI_PID_Compact_1".sPid_Calc.r_Cycle := 0.1; END_IF;
END_REGION

REGION Network 8: PID Compact Bon 2 - call technology block
   RUNG wire#powerrail
      "AI_PID_Compact_1".PID_Compact(Setpoint := "AI_PID_Bon2_SP", Input := "AI_TT3208_Bon2_Eff", Input_PER :=, ManualEnable := "AI_PID_Bon2_ManualEnable", ManualValue := "AI_PID_Bon2_ManualValue", Reset := "AI_PID_Bon2_Reset_Eff", ScaledInput =>, Output => "AI_PID_Bon2_CV", Output_PER =>, Output_PWM =>, SetpointLimit_H =>, SetpointLimit_L =>, InputWarning_H =>, InputWarning_L =>, State => "AI_PID_Bon2_State", Error => "AI_PID_Bon2_ErrorBits")
   END_RUNG
   // the same network as SCL:
   "AI_PID_Compact_1"(Setpoint := "AI_PID_Bon2_SP",   // PID_Compact
                      Input := "AI_TT3208_Bon2_Eff",
                      ManualEnable := "AI_PID_Bon2_ManualEnable",
                      ManualValue := "AI_PID_Bon2_ManualValue",
                      Reset := "AI_PID_Bon2_Reset_Eff",
                      Output => "AI_PID_Bon2_CV",
                      State => "AI_PID_Bon2_State",
                      Error => "AI_PID_Bon2_ErrorBits");
END_REGION

REGION Network 9: Detect PID Bon 2 Error
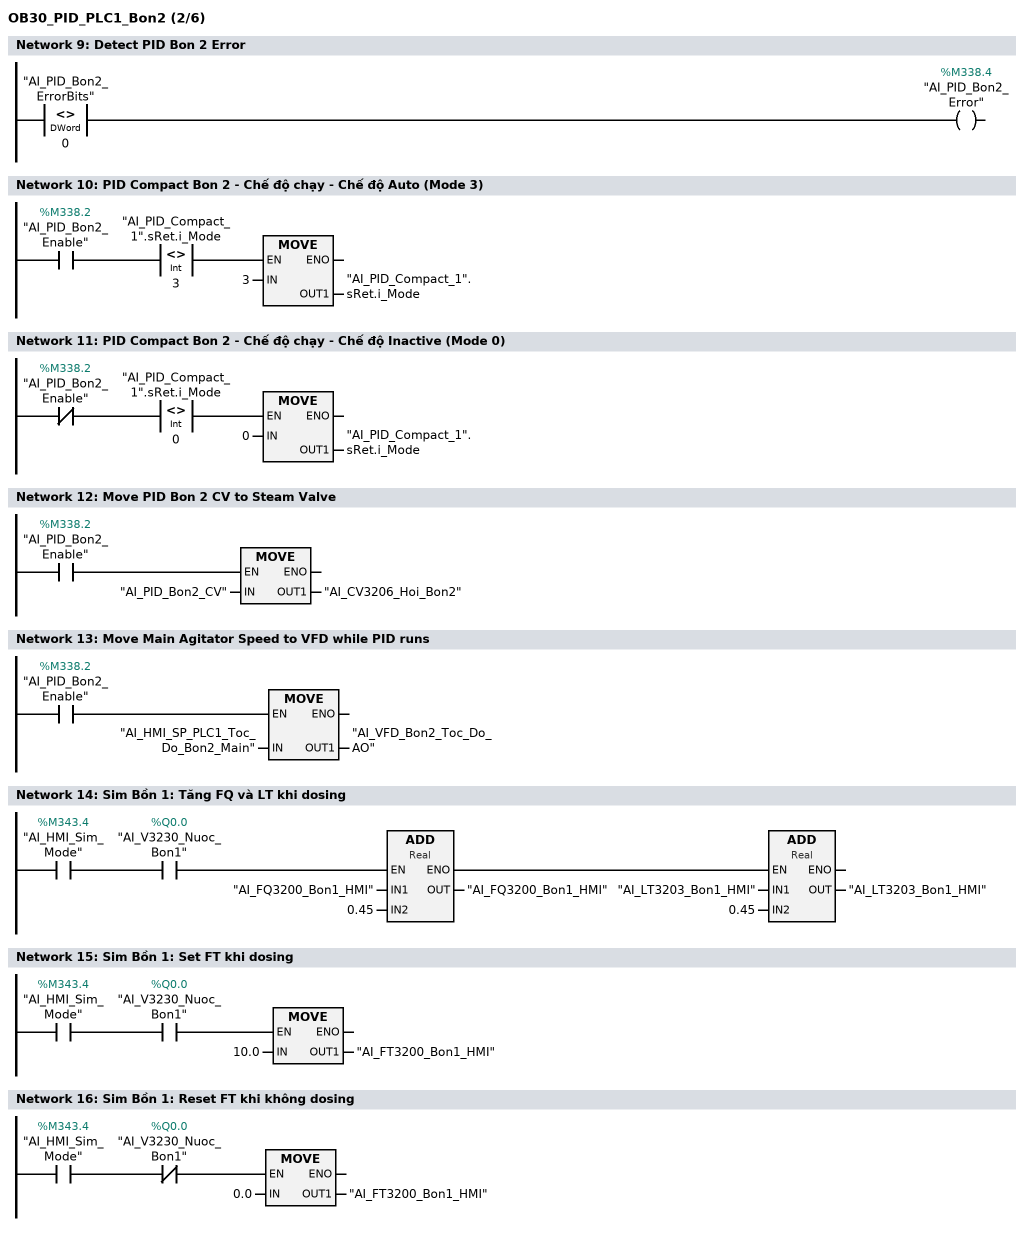
   RUNG wire#powerrail
      { S7_Templates := "SrcType := DWord" } NE_Contact(in1 := "AI_PID_Bon2_ErrorBits", in2 := 0)
      Coil( "AI_PID_Bon2_Error" )
   END_RUNG
   // the same network as SCL:
   "AI_PID_Bon2_Error" := "AI_PID_Bon2_ErrorBits" <> 0;
END_REGION

REGION Network 10: PID Compact Bon 2 - Chế độ chạy - Chế độ Auto (Mode 3)
   RUNG wire#powerrail
      Contact( "AI_PID_Bon2_Enable" )
      { S7_Templates := "SrcType := Int" } NE_Contact(in1 := "AI_PID_Compact_1".sRet.i_Mode, in2 := 3)
      { S7_GenerateENO := "TRUE" } Move(in := 3, out1 => "AI_PID_Compact_1".sRet.i_Mode)
   END_RUNG
   // the same network as SCL:
   IF "AI_PID_Bon2_Enable" AND ("AI_PID_Compact_1".sRet.i_Mode <> 3) THEN
       "AI_PID_Compact_1".sRet.i_Mode := 3;
   END_IF;
END_REGION

REGION Network 11: PID Compact Bon 2 - Chế độ chạy - Chế độ Inactive (Mode 0)
   RUNG wire#powerrail
      I_Contact( "AI_PID_Bon2_Enable" )
      { S7_Templates := "SrcType := Int" } NE_Contact(in1 := "AI_PID_Compact_1".sRet.i_Mode, in2 := 0)
      { S7_GenerateENO := "TRUE" } Move(in := 0, out1 => "AI_PID_Compact_1".sRet.i_Mode)
   END_RUNG
   // the same network as SCL:
   IF NOT "AI_PID_Bon2_Enable" AND ("AI_PID_Compact_1".sRet.i_Mode <> 0) THEN
       "AI_PID_Compact_1".sRet.i_Mode := 0;
   END_IF;
END_REGION

REGION Network 12: Move PID Bon 2 CV to Steam Valve
   RUNG wire#powerrail
      Contact( "AI_PID_Bon2_Enable" )
      { S7_GenerateENO := "TRUE" } Move(in := "AI_PID_Bon2_CV", out1 => "AI_CV3206_Hoi_Bon2")
   END_RUNG
   // the same network as SCL:
   IF "AI_PID_Bon2_Enable" THEN "AI_CV3206_Hoi_Bon2" := "AI_PID_Bon2_CV"; END_IF;
END_REGION

REGION Network 13: Move Main Agitator Speed to VFD while PID runs
   RUNG wire#powerrail
      Contact( "AI_PID_Bon2_Enable" )
      { S7_GenerateENO := "TRUE" } Move(in := "AI_HMI_SP_PLC1_Toc_Do_Bon2_Main", out1 => "AI_VFD_Bon2_Toc_Do_AO")
   END_RUNG
   // the same network as SCL:
   IF "AI_PID_Bon2_Enable" THEN "AI_VFD_Bon2_Toc_Do_AO" := "AI_HMI_SP_PLC1_Toc_Do_Bon2_Main"; END_IF;
END_REGION

REGION Network 14: Sim Bồn 1: Tăng FQ và LT khi dosing
   RUNG wire#powerrail
      Contact( "AI_HMI_Sim_Mode" )
      Contact( "AI_V3230_Nuoc_Bon1" )
      { S7_Templates := "SrcType := Real"; S7_GenerateENO := "TRUE" } Add(in1 := "AI_FQ3200_Bon1_HMI", in2 := 0.45, out => "AI_FQ3200_Bon1_HMI")
      { S7_Templates := "SrcType := Real"; S7_GenerateENO := "TRUE" } Add(in1 := "AI_LT3203_Bon1_HMI", in2 := 0.45, out => "AI_LT3203_Bon1_HMI")
   END_RUNG
   // the same network as SCL:
   // ENO of a box is taken as its EN; it also drops when the box reports an error
   IF "AI_HMI_Sim_Mode" AND "AI_V3230_Nuoc_Bon1" THEN
       "AI_FQ3200_Bon1_HMI" := "AI_FQ3200_Bon1_HMI" + 0.45;
       "AI_LT3203_Bon1_HMI" := "AI_LT3203_Bon1_HMI" + 0.45;
   END_IF;
END_REGION

REGION Network 15: Sim Bồn 1: Set FT khi dosing
   RUNG wire#powerrail
      Contact( "AI_HMI_Sim_Mode" )
      Contact( "AI_V3230_Nuoc_Bon1" )
      { S7_GenerateENO := "TRUE" } Move(in := 10.0, out1 => "AI_FT3200_Bon1_HMI")
   END_RUNG
   // the same network as SCL:
   IF "AI_HMI_Sim_Mode" AND "AI_V3230_Nuoc_Bon1" THEN "AI_FT3200_Bon1_HMI" := 10.0; END_IF;
END_REGION

REGION Network 16: Sim Bồn 1: Reset FT khi không dosing
   RUNG wire#powerrail
      Contact( "AI_HMI_Sim_Mode" )
      I_Contact( "AI_V3230_Nuoc_Bon1" )
      { S7_GenerateENO := "TRUE" } Move(in := 0.0, out1 => "AI_FT3200_Bon1_HMI")
   END_RUNG
   // the same network as SCL:
   IF "AI_HMI_Sim_Mode" AND NOT "AI_V3230_Nuoc_Bon1" THEN "AI_FT3200_Bon1_HMI" := 0.0; END_IF;
END_REGION

REGION Network 17: Sim Bồn 1: Giảm LT khi xả đáy
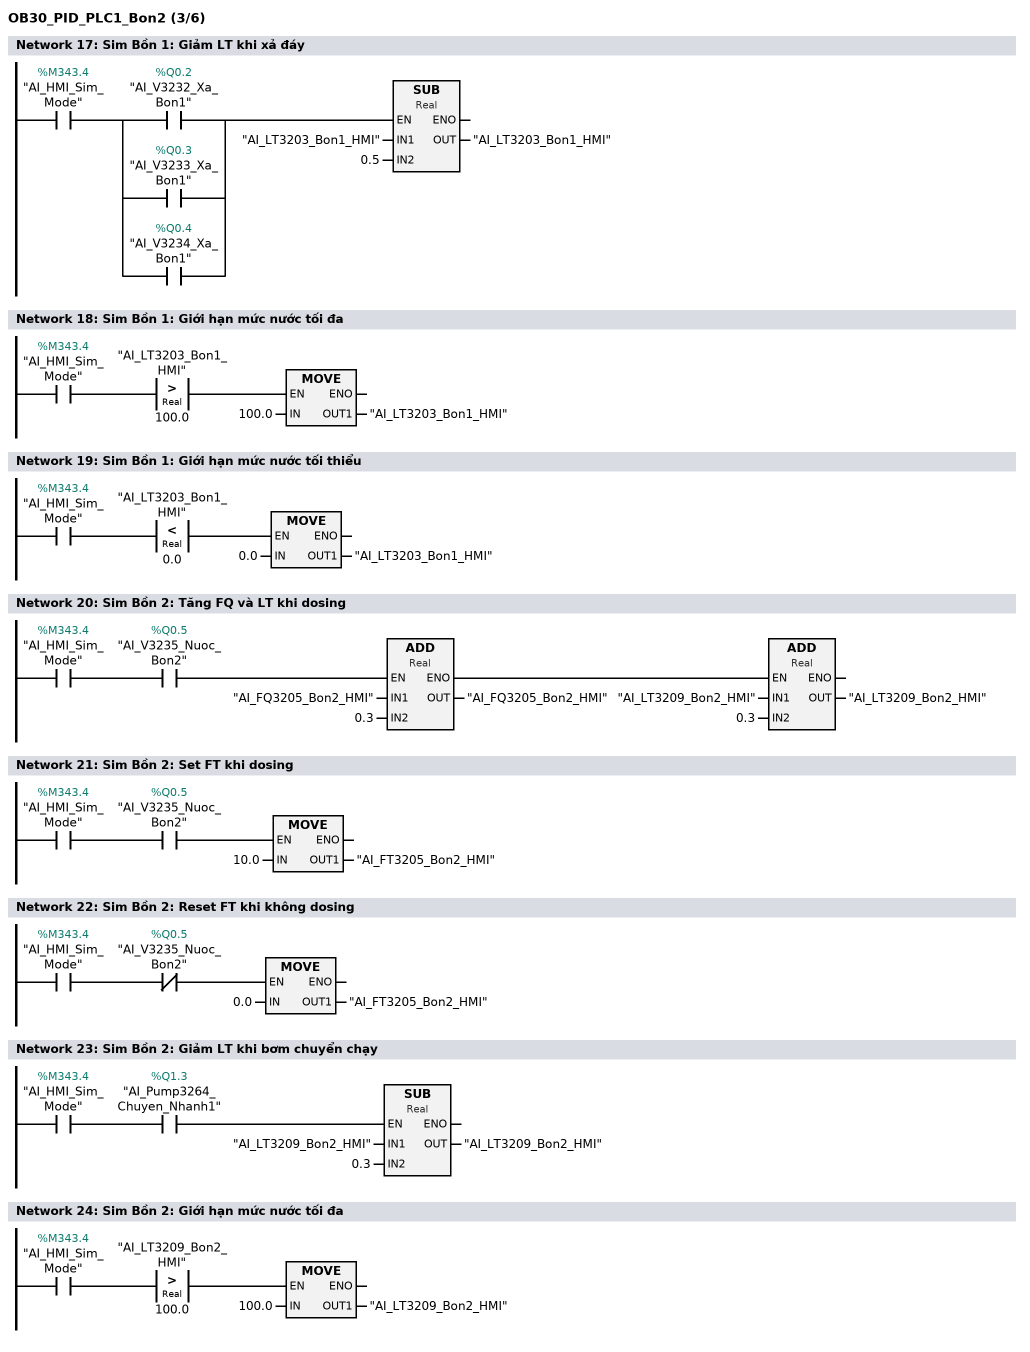
   RUNG wire#powerrail
      Contact( "AI_HMI_Sim_Mode" )
      wire#w1
      Contact( "AI_V3232_Xa_Bon1" )
      wire#w2
      { S7_Templates := "SrcType := Real"; S7_GenerateENO := "TRUE" } Sub(in1 := "AI_LT3203_Bon1_HMI", in2 := 0.5, out => "AI_LT3203_Bon1_HMI")
   END_RUNG
   RUNG wire#w1
      Contact( "AI_V3233_Xa_Bon1" )
   END_RUNG wire#w2
   RUNG wire#w1
      Contact( "AI_V3234_Xa_Bon1" )
   END_RUNG wire#w2
   // the same network as SCL:
   IF "AI_HMI_Sim_Mode" AND ("AI_V3232_Xa_Bon1" OR "AI_V3233_Xa_Bon1" OR "AI_V3234_Xa_Bon1") THEN
       "AI_LT3203_Bon1_HMI" := "AI_LT3203_Bon1_HMI" - 0.5;
   END_IF;
END_REGION

REGION Network 18: Sim Bồn 1: Giới hạn mức nước tối đa
   RUNG wire#powerrail
      Contact( "AI_HMI_Sim_Mode" )
      { S7_Templates := "SrcType := Real" } GT_Contact(in1 := "AI_LT3203_Bon1_HMI", in2 := 100.0)
      { S7_GenerateENO := "TRUE" } Move(in := 100.0, out1 => "AI_LT3203_Bon1_HMI")
   END_RUNG
   // the same network as SCL:
   IF "AI_HMI_Sim_Mode" AND ("AI_LT3203_Bon1_HMI" > 100.0) THEN "AI_LT3203_Bon1_HMI" := 100.0; END_IF;
END_REGION

REGION Network 19: Sim Bồn 1: Giới hạn mức nước tối thiểu
   RUNG wire#powerrail
      Contact( "AI_HMI_Sim_Mode" )
      { S7_Templates := "SrcType := Real" } LT_Contact(in1 := "AI_LT3203_Bon1_HMI", in2 := 0.0)
      { S7_GenerateENO := "TRUE" } Move(in := 0.0, out1 => "AI_LT3203_Bon1_HMI")
   END_RUNG
   // the same network as SCL:
   IF "AI_HMI_Sim_Mode" AND ("AI_LT3203_Bon1_HMI" < 0.0) THEN "AI_LT3203_Bon1_HMI" := 0.0; END_IF;
END_REGION

REGION Network 20: Sim Bồn 2: Tăng FQ và LT khi dosing
   RUNG wire#powerrail
      Contact( "AI_HMI_Sim_Mode" )
      Contact( "AI_V3235_Nuoc_Bon2" )
      { S7_Templates := "SrcType := Real"; S7_GenerateENO := "TRUE" } Add(in1 := "AI_FQ3205_Bon2_HMI", in2 := 0.3, out => "AI_FQ3205_Bon2_HMI")
      { S7_Templates := "SrcType := Real"; S7_GenerateENO := "TRUE" } Add(in1 := "AI_LT3209_Bon2_HMI", in2 := 0.3, out => "AI_LT3209_Bon2_HMI")
   END_RUNG
   // the same network as SCL:
   // ENO of a box is taken as its EN; it also drops when the box reports an error
   IF "AI_HMI_Sim_Mode" AND "AI_V3235_Nuoc_Bon2" THEN
       "AI_FQ3205_Bon2_HMI" := "AI_FQ3205_Bon2_HMI" + 0.3;
       "AI_LT3209_Bon2_HMI" := "AI_LT3209_Bon2_HMI" + 0.3;
   END_IF;
END_REGION

REGION Network 21: Sim Bồn 2: Set FT khi dosing
   RUNG wire#powerrail
      Contact( "AI_HMI_Sim_Mode" )
      Contact( "AI_V3235_Nuoc_Bon2" )
      { S7_GenerateENO := "TRUE" } Move(in := 10.0, out1 => "AI_FT3205_Bon2_HMI")
   END_RUNG
   // the same network as SCL:
   IF "AI_HMI_Sim_Mode" AND "AI_V3235_Nuoc_Bon2" THEN "AI_FT3205_Bon2_HMI" := 10.0; END_IF;
END_REGION

REGION Network 22: Sim Bồn 2: Reset FT khi không dosing
   RUNG wire#powerrail
      Contact( "AI_HMI_Sim_Mode" )
      I_Contact( "AI_V3235_Nuoc_Bon2" )
      { S7_GenerateENO := "TRUE" } Move(in := 0.0, out1 => "AI_FT3205_Bon2_HMI")
   END_RUNG
   // the same network as SCL:
   IF "AI_HMI_Sim_Mode" AND NOT "AI_V3235_Nuoc_Bon2" THEN "AI_FT3205_Bon2_HMI" := 0.0; END_IF;
END_REGION

REGION Network 23: Sim Bồn 2: Giảm LT khi bơm chuyển chạy
   RUNG wire#powerrail
      Contact( "AI_HMI_Sim_Mode" )
      Contact( "AI_Pump3264_Chuyen_Nhanh1" )
      { S7_Templates := "SrcType := Real"; S7_GenerateENO := "TRUE" } Sub(in1 := "AI_LT3209_Bon2_HMI", in2 := 0.3, out => "AI_LT3209_Bon2_HMI")
   END_RUNG
   // the same network as SCL:
   IF "AI_HMI_Sim_Mode" AND "AI_Pump3264_Chuyen_Nhanh1" THEN
       "AI_LT3209_Bon2_HMI" := "AI_LT3209_Bon2_HMI" - 0.3;
   END_IF;
END_REGION

REGION Network 24: Sim Bồn 2: Giới hạn mức nước tối đa
   RUNG wire#powerrail
      Contact( "AI_HMI_Sim_Mode" )
      { S7_Templates := "SrcType := Real" } GT_Contact(in1 := "AI_LT3209_Bon2_HMI", in2 := 100.0)
      { S7_GenerateENO := "TRUE" } Move(in := 100.0, out1 => "AI_LT3209_Bon2_HMI")
   END_RUNG
   // the same network as SCL:
   IF "AI_HMI_Sim_Mode" AND ("AI_LT3209_Bon2_HMI" > 100.0) THEN "AI_LT3209_Bon2_HMI" := 100.0; END_IF;
END_REGION

REGION Network 25: Sim Bồn 2: Giới hạn mức nước tối thiểu
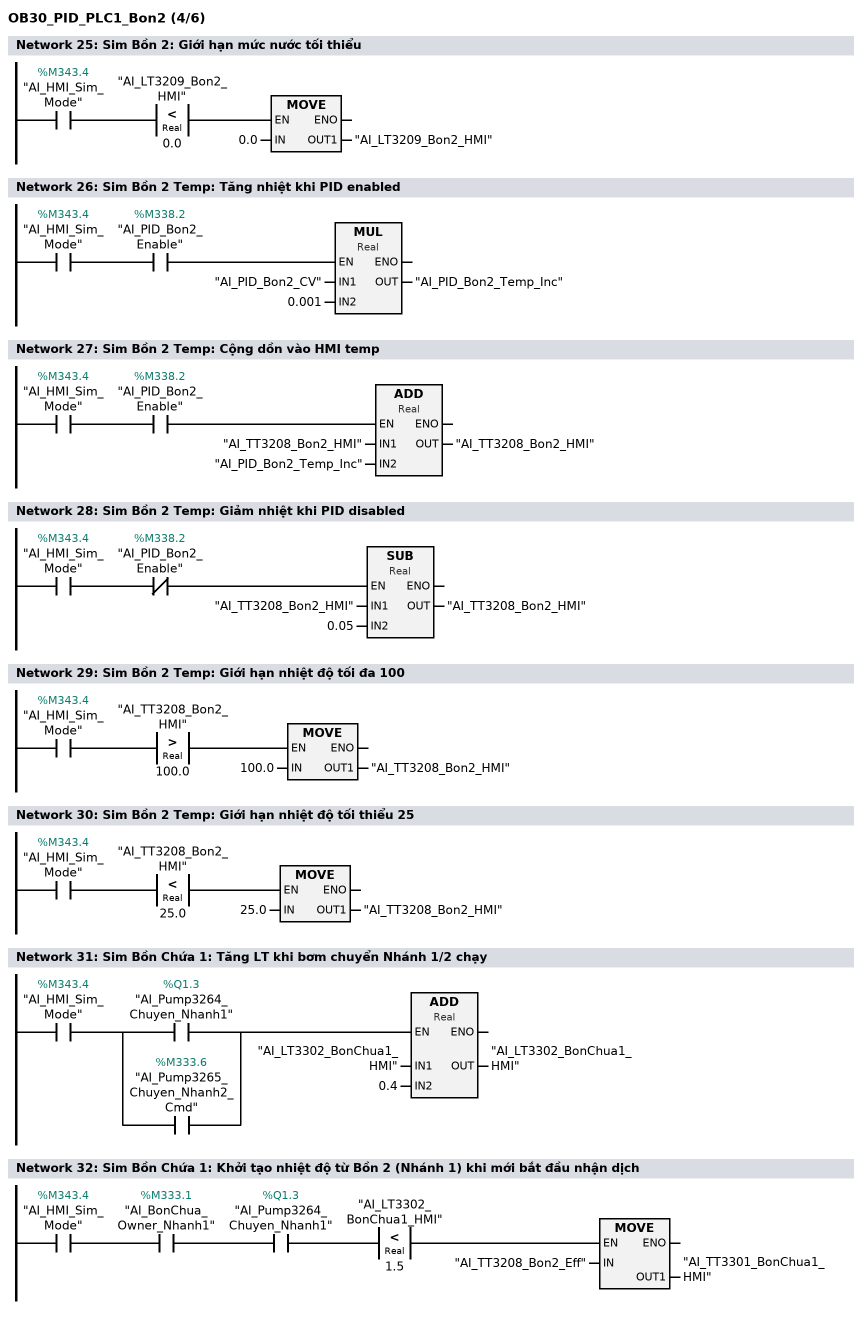
   RUNG wire#powerrail
      Contact( "AI_HMI_Sim_Mode" )
      { S7_Templates := "SrcType := Real" } LT_Contact(in1 := "AI_LT3209_Bon2_HMI", in2 := 0.0)
      { S7_GenerateENO := "TRUE" } Move(in := 0.0, out1 => "AI_LT3209_Bon2_HMI")
   END_RUNG
   // the same network as SCL:
   IF "AI_HMI_Sim_Mode" AND ("AI_LT3209_Bon2_HMI" < 0.0) THEN "AI_LT3209_Bon2_HMI" := 0.0; END_IF;
END_REGION

REGION Network 26: Sim Bồn 2 Temp: Tăng nhiệt khi PID enabled
   RUNG wire#powerrail
      Contact( "AI_HMI_Sim_Mode" )
      Contact( "AI_PID_Bon2_Enable" )
      { S7_Templates := "SrcType := Real"; S7_GenerateENO := "TRUE" } Mul(in1 := "AI_PID_Bon2_CV", in2 := 0.001, out => "AI_PID_Bon2_Temp_Inc")
   END_RUNG
   // the same network as SCL:
   IF "AI_HMI_Sim_Mode" AND "AI_PID_Bon2_Enable" THEN
       "AI_PID_Bon2_Temp_Inc" := "AI_PID_Bon2_CV" * 0.001;
   END_IF;
END_REGION

REGION Network 27: Sim Bồn 2 Temp: Cộng dồn vào HMI temp
   RUNG wire#powerrail
      Contact( "AI_HMI_Sim_Mode" )
      Contact( "AI_PID_Bon2_Enable" )
      { S7_Templates := "SrcType := Real"; S7_GenerateENO := "TRUE" } Add(in1 := "AI_TT3208_Bon2_HMI", in2 := "AI_PID_Bon2_Temp_Inc", out => "AI_TT3208_Bon2_HMI")
   END_RUNG
   // the same network as SCL:
   IF "AI_HMI_Sim_Mode" AND "AI_PID_Bon2_Enable" THEN
       "AI_TT3208_Bon2_HMI" := "AI_TT3208_Bon2_HMI" + "AI_PID_Bon2_Temp_Inc";
   END_IF;
END_REGION

REGION Network 28: Sim Bồn 2 Temp: Giảm nhiệt khi PID disabled
   RUNG wire#powerrail
      Contact( "AI_HMI_Sim_Mode" )
      I_Contact( "AI_PID_Bon2_Enable" )
      { S7_Templates := "SrcType := Real"; S7_GenerateENO := "TRUE" } Sub(in1 := "AI_TT3208_Bon2_HMI", in2 := 0.05, out => "AI_TT3208_Bon2_HMI")
   END_RUNG
   // the same network as SCL:
   IF "AI_HMI_Sim_Mode" AND NOT "AI_PID_Bon2_Enable" THEN
       "AI_TT3208_Bon2_HMI" := "AI_TT3208_Bon2_HMI" - 0.05;
   END_IF;
END_REGION

REGION Network 29: Sim Bồn 2 Temp: Giới hạn nhiệt độ tối đa 100
   RUNG wire#powerrail
      Contact( "AI_HMI_Sim_Mode" )
      { S7_Templates := "SrcType := Real" } GT_Contact(in1 := "AI_TT3208_Bon2_HMI", in2 := 100.0)
      { S7_GenerateENO := "TRUE" } Move(in := 100.0, out1 => "AI_TT3208_Bon2_HMI")
   END_RUNG
   // the same network as SCL:
   IF "AI_HMI_Sim_Mode" AND ("AI_TT3208_Bon2_HMI" > 100.0) THEN "AI_TT3208_Bon2_HMI" := 100.0; END_IF;
END_REGION

REGION Network 30: Sim Bồn 2 Temp: Giới hạn nhiệt độ tối thiểu 25
   RUNG wire#powerrail
      Contact( "AI_HMI_Sim_Mode" )
      { S7_Templates := "SrcType := Real" } LT_Contact(in1 := "AI_TT3208_Bon2_HMI", in2 := 25.0)
      { S7_GenerateENO := "TRUE" } Move(in := 25.0, out1 => "AI_TT3208_Bon2_HMI")
   END_RUNG
   // the same network as SCL:
   IF "AI_HMI_Sim_Mode" AND ("AI_TT3208_Bon2_HMI" < 25.0) THEN "AI_TT3208_Bon2_HMI" := 25.0; END_IF;
END_REGION

REGION Network 31: Sim Bồn Chứa 1: Tăng LT khi bơm chuyển Nhánh 1/2 chạy
   RUNG wire#powerrail
      Contact( "AI_HMI_Sim_Mode" )
      wire#w1
      Contact( "AI_Pump3264_Chuyen_Nhanh1" )
      wire#w2
      { S7_Templates := "SrcType := Real"; S7_GenerateENO := "TRUE" } Add(in1 := "AI_LT3302_BonChua1_HMI", in2 := 0.4, out => "AI_LT3302_BonChua1_HMI")
   END_RUNG
   RUNG wire#w1
      Contact( "AI_Pump3265_Chuyen_Nhanh2_Cmd" )
   END_RUNG wire#w2
   // the same network as SCL:
   IF "AI_HMI_Sim_Mode" AND ("AI_Pump3264_Chuyen_Nhanh1" OR "AI_Pump3265_Chuyen_Nhanh2_Cmd") THEN
       "AI_LT3302_BonChua1_HMI" := "AI_LT3302_BonChua1_HMI" + 0.4;
   END_IF;
END_REGION

REGION Network 32: Sim Bồn Chứa 1: Khởi tạo nhiệt độ từ Bồn 2 (Nhánh 1) khi mới bắt đầu nhận dịch
   RUNG wire#powerrail
      Contact( "AI_HMI_Sim_Mode" )
      Contact( "AI_BonChua_Owner_Nhanh1" )
      Contact( "AI_Pump3264_Chuyen_Nhanh1" )
      { S7_Templates := "SrcType := Real" } LT_Contact(in1 := "AI_LT3302_BonChua1_HMI", in2 := 1.5)
      { S7_GenerateENO := "TRUE" } Move(in := "AI_TT3208_Bon2_Eff", out1 => "AI_TT3301_BonChua1_HMI")
   END_RUNG
   // the same network as SCL:
   IF "AI_HMI_Sim_Mode" AND "AI_BonChua_Owner_Nhanh1" AND "AI_Pump3264_Chuyen_Nhanh1" AND ("AI_LT3302_BonChua1_HMI" < 1.5) THEN
       "AI_TT3301_BonChua1_HMI" := "AI_TT3208_Bon2_Eff";
   END_IF;
END_REGION

REGION Network 33: Sim Bồn Chứa 1: Khởi tạo nhiệt độ từ Bồn 4 (Nhánh 2) khi mới bắt đầu nhận dịch
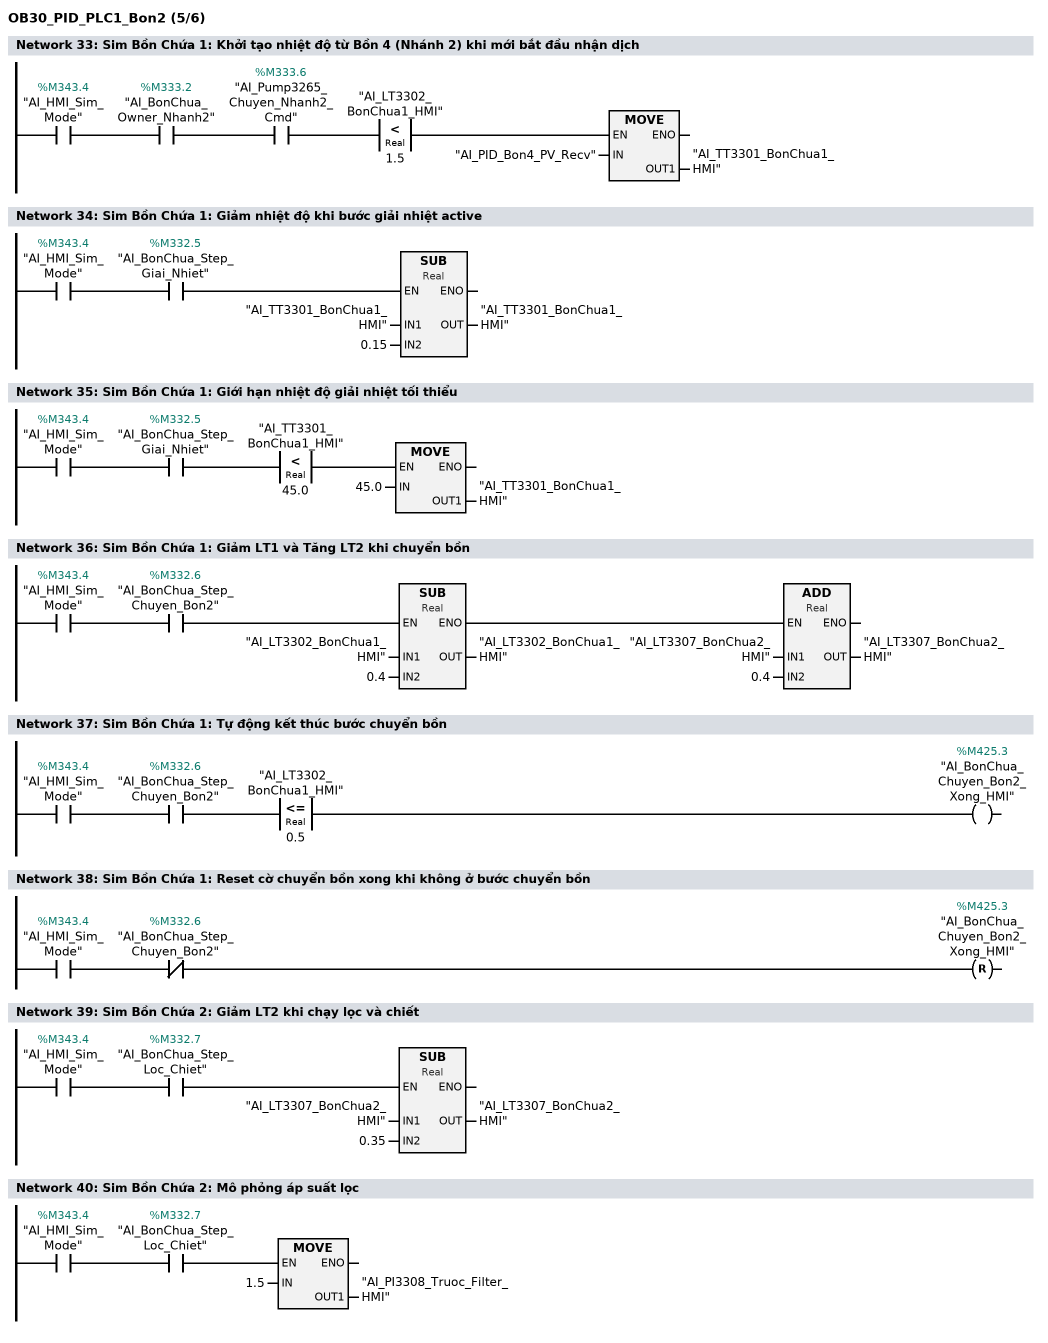
   RUNG wire#powerrail
      Contact( "AI_HMI_Sim_Mode" )
      Contact( "AI_BonChua_Owner_Nhanh2" )
      Contact( "AI_Pump3265_Chuyen_Nhanh2_Cmd" )
      { S7_Templates := "SrcType := Real" } LT_Contact(in1 := "AI_LT3302_BonChua1_HMI", in2 := 1.5)
      { S7_GenerateENO := "TRUE" } Move(in := "AI_PID_Bon4_PV_Recv", out1 => "AI_TT3301_BonChua1_HMI")
   END_RUNG
   // the same network as SCL:
   IF "AI_HMI_Sim_Mode" AND "AI_BonChua_Owner_Nhanh2" AND "AI_Pump3265_Chuyen_Nhanh2_Cmd" AND ("AI_LT3302_BonChua1_HMI" < 1.5) THEN
       "AI_TT3301_BonChua1_HMI" := "AI_PID_Bon4_PV_Recv";
   END_IF;
END_REGION

REGION Network 34: Sim Bồn Chứa 1: Giảm nhiệt độ khi bước giải nhiệt active
   RUNG wire#powerrail
      Contact( "AI_HMI_Sim_Mode" )
      Contact( "AI_BonChua_Step_Giai_Nhiet" )
      { S7_Templates := "SrcType := Real"; S7_GenerateENO := "TRUE" } Sub(in1 := "AI_TT3301_BonChua1_HMI", in2 := 0.15, out => "AI_TT3301_BonChua1_HMI")
   END_RUNG
   // the same network as SCL:
   IF "AI_HMI_Sim_Mode" AND "AI_BonChua_Step_Giai_Nhiet" THEN
       "AI_TT3301_BonChua1_HMI" := "AI_TT3301_BonChua1_HMI" - 0.15;
   END_IF;
END_REGION

REGION Network 35: Sim Bồn Chứa 1: Giới hạn nhiệt độ giải nhiệt tối thiểu
   RUNG wire#powerrail
      Contact( "AI_HMI_Sim_Mode" )
      Contact( "AI_BonChua_Step_Giai_Nhiet" )
      { S7_Templates := "SrcType := Real" } LT_Contact(in1 := "AI_TT3301_BonChua1_HMI", in2 := 45.0)
      { S7_GenerateENO := "TRUE" } Move(in := 45.0, out1 => "AI_TT3301_BonChua1_HMI")
   END_RUNG
   // the same network as SCL:
   IF "AI_HMI_Sim_Mode" AND "AI_BonChua_Step_Giai_Nhiet" AND ("AI_TT3301_BonChua1_HMI" < 45.0) THEN
       "AI_TT3301_BonChua1_HMI" := 45.0;
   END_IF;
END_REGION

REGION Network 36: Sim Bồn Chứa 1: Giảm LT1 và Tăng LT2 khi chuyển bồn
   RUNG wire#powerrail
      Contact( "AI_HMI_Sim_Mode" )
      Contact( "AI_BonChua_Step_Chuyen_Bon2" )
      { S7_Templates := "SrcType := Real"; S7_GenerateENO := "TRUE" } Sub(in1 := "AI_LT3302_BonChua1_HMI", in2 := 0.4, out => "AI_LT3302_BonChua1_HMI")
      { S7_Templates := "SrcType := Real"; S7_GenerateENO := "TRUE" } Add(in1 := "AI_LT3307_BonChua2_HMI", in2 := 0.4, out => "AI_LT3307_BonChua2_HMI")
   END_RUNG
   // the same network as SCL:
   // ENO of a box is taken as its EN; it also drops when the box reports an error
   IF "AI_HMI_Sim_Mode" AND "AI_BonChua_Step_Chuyen_Bon2" THEN
       "AI_LT3302_BonChua1_HMI" := "AI_LT3302_BonChua1_HMI" - 0.4;
       "AI_LT3307_BonChua2_HMI" := "AI_LT3307_BonChua2_HMI" + 0.4;
   END_IF;
END_REGION

REGION Network 37: Sim Bồn Chứa 1: Tự động kết thúc bước chuyển bồn
   RUNG wire#powerrail
      Contact( "AI_HMI_Sim_Mode" )
      Contact( "AI_BonChua_Step_Chuyen_Bon2" )
      { S7_Templates := "SrcType := Real" } LE_Contact(in1 := "AI_LT3302_BonChua1_HMI", in2 := 0.5)
      Coil( "AI_BonChua_Chuyen_Bon2_Xong_HMI" )
   END_RUNG
   // the same network as SCL:
   "AI_BonChua_Chuyen_Bon2_Xong_HMI" := "AI_HMI_Sim_Mode" AND "AI_BonChua_Step_Chuyen_Bon2" AND ("AI_LT3302_BonChua1_HMI" <= 0.5);
END_REGION

REGION Network 38: Sim Bồn Chứa 1: Reset cờ chuyển bồn xong khi không ở bước chuyển bồn
   RUNG wire#powerrail
      Contact( "AI_HMI_Sim_Mode" )
      I_Contact( "AI_BonChua_Step_Chuyen_Bon2" )
      R_Coil( "AI_BonChua_Chuyen_Bon2_Xong_HMI" )
   END_RUNG
   // the same network as SCL:
   IF "AI_HMI_Sim_Mode" AND NOT "AI_BonChua_Step_Chuyen_Bon2" THEN
       "AI_BonChua_Chuyen_Bon2_Xong_HMI" := FALSE;
   END_IF;
END_REGION

REGION Network 39: Sim Bồn Chứa 2: Giảm LT2 khi chạy lọc và chiết
   RUNG wire#powerrail
      Contact( "AI_HMI_Sim_Mode" )
      Contact( "AI_BonChua_Step_Loc_Chiet" )
      { S7_Templates := "SrcType := Real"; S7_GenerateENO := "TRUE" } Sub(in1 := "AI_LT3307_BonChua2_HMI", in2 := 0.35, out => "AI_LT3307_BonChua2_HMI")
   END_RUNG
   // the same network as SCL:
   IF "AI_HMI_Sim_Mode" AND "AI_BonChua_Step_Loc_Chiet" THEN
       "AI_LT3307_BonChua2_HMI" := "AI_LT3307_BonChua2_HMI" - 0.35;
   END_IF;
END_REGION

REGION Network 40: Sim Bồn Chứa 2: Mô phỏng áp suất lọc
   RUNG wire#powerrail
      Contact( "AI_HMI_Sim_Mode" )
      Contact( "AI_BonChua_Step_Loc_Chiet" )
      { S7_GenerateENO := "TRUE" } Move(in := 1.5, out1 => "AI_PI3308_Truoc_Filter_HMI")
   END_RUNG
   // the same network as SCL:
   IF "AI_HMI_Sim_Mode" AND "AI_BonChua_Step_Loc_Chiet" THEN "AI_PI3308_Truoc_Filter_HMI" := 1.5; END_IF;
END_REGION

REGION Network 41: Sim Bồn Chứa 2: Mô phỏng lưu lượng xả
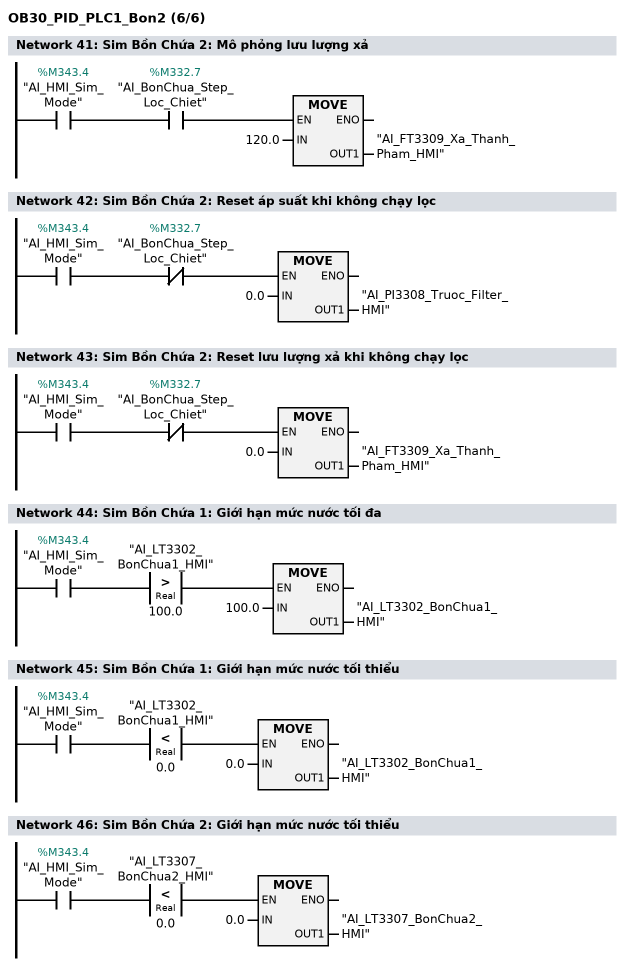
   RUNG wire#powerrail
      Contact( "AI_HMI_Sim_Mode" )
      Contact( "AI_BonChua_Step_Loc_Chiet" )
      { S7_GenerateENO := "TRUE" } Move(in := 120.0, out1 => "AI_FT3309_Xa_Thanh_Pham_HMI")
   END_RUNG
   // the same network as SCL:
   IF "AI_HMI_Sim_Mode" AND "AI_BonChua_Step_Loc_Chiet" THEN "AI_FT3309_Xa_Thanh_Pham_HMI" := 120.0; END_IF;
END_REGION

REGION Network 42: Sim Bồn Chứa 2: Reset áp suất khi không chạy lọc
   RUNG wire#powerrail
      Contact( "AI_HMI_Sim_Mode" )
      I_Contact( "AI_BonChua_Step_Loc_Chiet" )
      { S7_GenerateENO := "TRUE" } Move(in := 0.0, out1 => "AI_PI3308_Truoc_Filter_HMI")
   END_RUNG
   // the same network as SCL:
   IF "AI_HMI_Sim_Mode" AND NOT "AI_BonChua_Step_Loc_Chiet" THEN "AI_PI3308_Truoc_Filter_HMI" := 0.0; END_IF;
END_REGION

REGION Network 43: Sim Bồn Chứa 2: Reset lưu lượng xả khi không chạy lọc
   RUNG wire#powerrail
      Contact( "AI_HMI_Sim_Mode" )
      I_Contact( "AI_BonChua_Step_Loc_Chiet" )
      { S7_GenerateENO := "TRUE" } Move(in := 0.0, out1 => "AI_FT3309_Xa_Thanh_Pham_HMI")
   END_RUNG
   // the same network as SCL:
   IF "AI_HMI_Sim_Mode" AND NOT "AI_BonChua_Step_Loc_Chiet" THEN
       "AI_FT3309_Xa_Thanh_Pham_HMI" := 0.0;
   END_IF;
END_REGION

REGION Network 44: Sim Bồn Chứa 1: Giới hạn mức nước tối đa
   RUNG wire#powerrail
      Contact( "AI_HMI_Sim_Mode" )
      { S7_Templates := "SrcType := Real" } GT_Contact(in1 := "AI_LT3302_BonChua1_HMI", in2 := 100.0)
      { S7_GenerateENO := "TRUE" } Move(in := 100.0, out1 => "AI_LT3302_BonChua1_HMI")
   END_RUNG
   // the same network as SCL:
   IF "AI_HMI_Sim_Mode" AND ("AI_LT3302_BonChua1_HMI" > 100.0) THEN
       "AI_LT3302_BonChua1_HMI" := 100.0;
   END_IF;
END_REGION

REGION Network 45: Sim Bồn Chứa 1: Giới hạn mức nước tối thiểu
   RUNG wire#powerrail
      Contact( "AI_HMI_Sim_Mode" )
      { S7_Templates := "SrcType := Real" } LT_Contact(in1 := "AI_LT3302_BonChua1_HMI", in2 := 0.0)
      { S7_GenerateENO := "TRUE" } Move(in := 0.0, out1 => "AI_LT3302_BonChua1_HMI")
   END_RUNG
   // the same network as SCL:
   IF "AI_HMI_Sim_Mode" AND ("AI_LT3302_BonChua1_HMI" < 0.0) THEN "AI_LT3302_BonChua1_HMI" := 0.0; END_IF;
END_REGION

REGION Network 46: Sim Bồn Chứa 2: Giới hạn mức nước tối thiểu
   RUNG wire#powerrail
      Contact( "AI_HMI_Sim_Mode" )
      { S7_Templates := "SrcType := Real" } LT_Contact(in1 := "AI_LT3307_BonChua2_HMI", in2 := 0.0)
      { S7_GenerateENO := "TRUE" } Move(in := 0.0, out1 => "AI_LT3307_BonChua2_HMI")
   END_RUNG
   // the same network as SCL:
   IF "AI_HMI_Sim_Mode" AND ("AI_LT3307_BonChua2_HMI" < 0.0) THEN "AI_LT3307_BonChua2_HMI" := 0.0; END_IF;
END_REGION
END_ORGANIZATION_BLOCK

ORGANIZATION_BLOCK "OB31_PID_PLC2_Bon4"   // OB31, LAD, CyclicInterrupt
{ S7_Optimized_Access := 'TRUE' }
VERSION : 0.1
// stored: AutoNumber true, IsIECCheckEnabled false
   VAR_INPUT
      Initial_Call : Bool;
      Remanence : Bool;
   END_VAR
BEGIN

REGION Network 1: Initialize PID Bon 4 Kp parameter
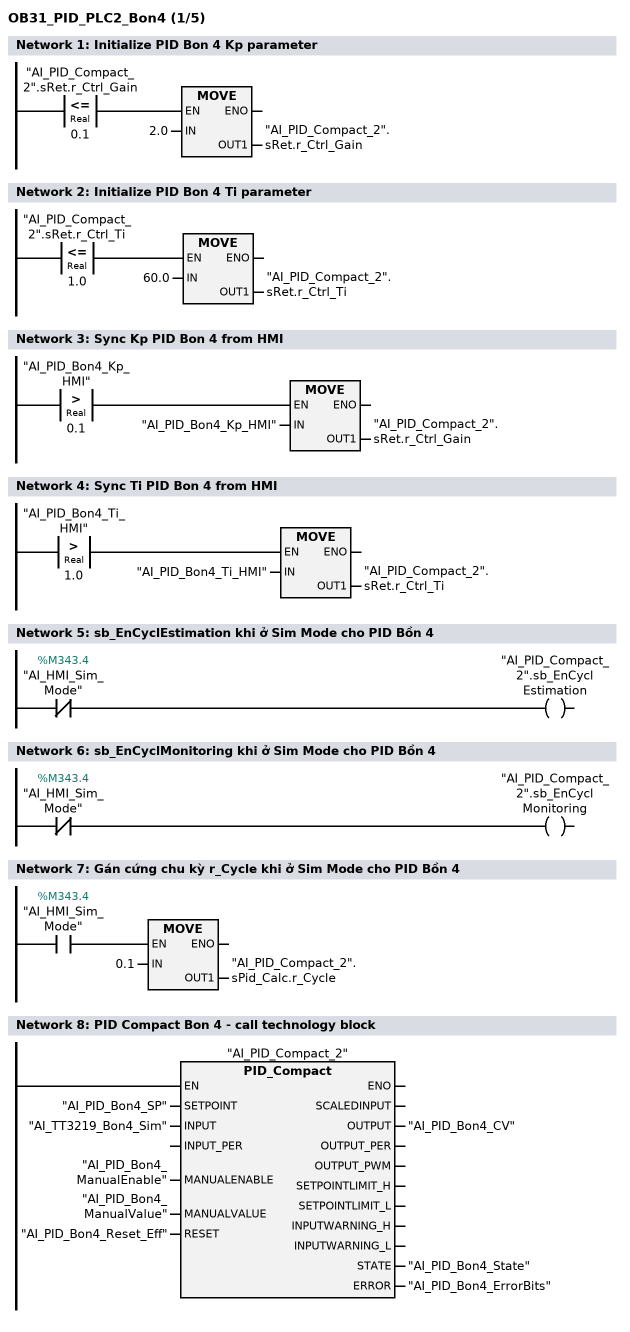
   RUNG wire#powerrail
      { S7_Templates := "SrcType := Real" } LE_Contact(in1 := "AI_PID_Compact_2".sRet.r_Ctrl_Gain, in2 := 0.1)
      { S7_GenerateENO := "TRUE" } Move(in := 2.0, out1 => "AI_PID_Compact_2".sRet.r_Ctrl_Gain)
   END_RUNG
   // the same network as SCL:
   IF "AI_PID_Compact_2".sRet.r_Ctrl_Gain <= 0.1 THEN "AI_PID_Compact_2".sRet.r_Ctrl_Gain := 2.0; END_IF;
END_REGION

REGION Network 2: Initialize PID Bon 4 Ti parameter
   RUNG wire#powerrail
      { S7_Templates := "SrcType := Real" } LE_Contact(in1 := "AI_PID_Compact_2".sRet.r_Ctrl_Ti, in2 := 1.0)
      { S7_GenerateENO := "TRUE" } Move(in := 60.0, out1 => "AI_PID_Compact_2".sRet.r_Ctrl_Ti)
   END_RUNG
   // the same network as SCL:
   IF "AI_PID_Compact_2".sRet.r_Ctrl_Ti <= 1.0 THEN "AI_PID_Compact_2".sRet.r_Ctrl_Ti := 60.0; END_IF;
END_REGION

REGION Network 3: Sync Kp PID Bon 4 from HMI
   RUNG wire#powerrail
      { S7_Templates := "SrcType := Real" } GT_Contact(in1 := "AI_PID_Bon4_Kp_HMI", in2 := 0.1)
      { S7_GenerateENO := "TRUE" } Move(in := "AI_PID_Bon4_Kp_HMI", out1 => "AI_PID_Compact_2".sRet.r_Ctrl_Gain)
   END_RUNG
   // the same network as SCL:
   IF "AI_PID_Bon4_Kp_HMI" > 0.1 THEN "AI_PID_Compact_2".sRet.r_Ctrl_Gain := "AI_PID_Bon4_Kp_HMI"; END_IF;
END_REGION

REGION Network 4: Sync Ti PID Bon 4 from HMI
   RUNG wire#powerrail
      { S7_Templates := "SrcType := Real" } GT_Contact(in1 := "AI_PID_Bon4_Ti_HMI", in2 := 1.0)
      { S7_GenerateENO := "TRUE" } Move(in := "AI_PID_Bon4_Ti_HMI", out1 => "AI_PID_Compact_2".sRet.r_Ctrl_Ti)
   END_RUNG
   // the same network as SCL:
   IF "AI_PID_Bon4_Ti_HMI" > 1.0 THEN "AI_PID_Compact_2".sRet.r_Ctrl_Ti := "AI_PID_Bon4_Ti_HMI"; END_IF;
END_REGION

REGION Network 5: sb_EnCyclEstimation khi ở Sim Mode cho PID Bồn 4
   RUNG wire#powerrail
      I_Contact( "AI_HMI_Sim_Mode" )
      Coil( "AI_PID_Compact_2".sb_EnCyclEstimation )
   END_RUNG
   // the same network as SCL:
   "AI_PID_Compact_2".sb_EnCyclEstimation := NOT "AI_HMI_Sim_Mode";
END_REGION

REGION Network 6: sb_EnCyclMonitoring khi ở Sim Mode cho PID Bồn 4
   RUNG wire#powerrail
      I_Contact( "AI_HMI_Sim_Mode" )
      Coil( "AI_PID_Compact_2".sb_EnCyclMonitoring )
   END_RUNG
   // the same network as SCL:
   "AI_PID_Compact_2".sb_EnCyclMonitoring := NOT "AI_HMI_Sim_Mode";
END_REGION

REGION Network 7: Gán cứng chu kỳ r_Cycle khi ở Sim Mode cho PID Bồn 4
   RUNG wire#powerrail
      Contact( "AI_HMI_Sim_Mode" )
      { S7_GenerateENO := "TRUE" } Move(in := 0.1, out1 => "AI_PID_Compact_2".sPid_Calc.r_Cycle)
   END_RUNG
   // the same network as SCL:
   IF "AI_HMI_Sim_Mode" THEN "AI_PID_Compact_2".sPid_Calc.r_Cycle := 0.1; END_IF;
END_REGION

REGION Network 8: PID Compact Bon 4 - call technology block
   RUNG wire#powerrail
      "AI_PID_Compact_2".PID_Compact(Setpoint := "AI_PID_Bon4_SP", Input := "AI_TT3219_Bon4_Sim", Input_PER :=, ManualEnable := "AI_PID_Bon4_ManualEnable", ManualValue := "AI_PID_Bon4_ManualValue", Reset := "AI_PID_Bon4_Reset_Eff", ScaledInput =>, Output => "AI_PID_Bon4_CV", Output_PER =>, Output_PWM =>, SetpointLimit_H =>, SetpointLimit_L =>, InputWarning_H =>, InputWarning_L =>, State => "AI_PID_Bon4_State", Error => "AI_PID_Bon4_ErrorBits")
   END_RUNG
   // the same network as SCL:
   "AI_PID_Compact_2"(Setpoint := "AI_PID_Bon4_SP",   // PID_Compact
                      Input := "AI_TT3219_Bon4_Sim",
                      ManualEnable := "AI_PID_Bon4_ManualEnable",
                      ManualValue := "AI_PID_Bon4_ManualValue",
                      Reset := "AI_PID_Bon4_Reset_Eff",
                      Output => "AI_PID_Bon4_CV",
                      State => "AI_PID_Bon4_State",
                      Error => "AI_PID_Bon4_ErrorBits");
END_REGION

REGION Network 9: Detect PID Bon 4 Error
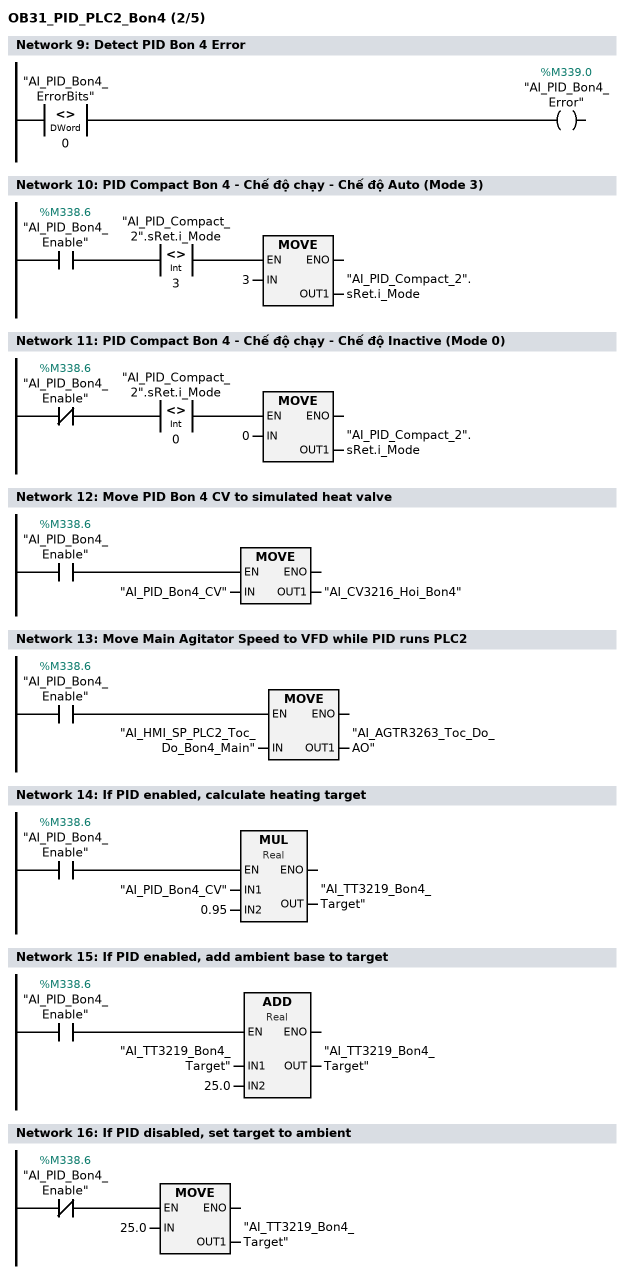
   RUNG wire#powerrail
      { S7_Templates := "SrcType := DWord" } NE_Contact(in1 := "AI_PID_Bon4_ErrorBits", in2 := 0)
      Coil( "AI_PID_Bon4_Error" )
   END_RUNG
   // the same network as SCL:
   "AI_PID_Bon4_Error" := "AI_PID_Bon4_ErrorBits" <> 0;
END_REGION

REGION Network 10: PID Compact Bon 4 - Chế độ chạy - Chế độ Auto (Mode 3)
   RUNG wire#powerrail
      Contact( "AI_PID_Bon4_Enable" )
      { S7_Templates := "SrcType := Int" } NE_Contact(in1 := "AI_PID_Compact_2".sRet.i_Mode, in2 := 3)
      { S7_GenerateENO := "TRUE" } Move(in := 3, out1 => "AI_PID_Compact_2".sRet.i_Mode)
   END_RUNG
   // the same network as SCL:
   IF "AI_PID_Bon4_Enable" AND ("AI_PID_Compact_2".sRet.i_Mode <> 3) THEN
       "AI_PID_Compact_2".sRet.i_Mode := 3;
   END_IF;
END_REGION

REGION Network 11: PID Compact Bon 4 - Chế độ chạy - Chế độ Inactive (Mode 0)
   RUNG wire#powerrail
      I_Contact( "AI_PID_Bon4_Enable" )
      { S7_Templates := "SrcType := Int" } NE_Contact(in1 := "AI_PID_Compact_2".sRet.i_Mode, in2 := 0)
      { S7_GenerateENO := "TRUE" } Move(in := 0, out1 => "AI_PID_Compact_2".sRet.i_Mode)
   END_RUNG
   // the same network as SCL:
   IF NOT "AI_PID_Bon4_Enable" AND ("AI_PID_Compact_2".sRet.i_Mode <> 0) THEN
       "AI_PID_Compact_2".sRet.i_Mode := 0;
   END_IF;
END_REGION

REGION Network 12: Move PID Bon 4 CV to simulated heat valve
   RUNG wire#powerrail
      Contact( "AI_PID_Bon4_Enable" )
      { S7_GenerateENO := "TRUE" } Move(in := "AI_PID_Bon4_CV", out1 => "AI_CV3216_Hoi_Bon4")
   END_RUNG
   // the same network as SCL:
   IF "AI_PID_Bon4_Enable" THEN "AI_CV3216_Hoi_Bon4" := "AI_PID_Bon4_CV"; END_IF;
END_REGION

REGION Network 13: Move Main Agitator Speed to VFD while PID runs PLC2
   RUNG wire#powerrail
      Contact( "AI_PID_Bon4_Enable" )
      { S7_GenerateENO := "TRUE" } Move(in := "AI_HMI_SP_PLC2_Toc_Do_Bon4_Main", out1 => "AI_AGTR3263_Toc_Do_AO")
   END_RUNG
   // the same network as SCL:
   IF "AI_PID_Bon4_Enable" THEN "AI_AGTR3263_Toc_Do_AO" := "AI_HMI_SP_PLC2_Toc_Do_Bon4_Main"; END_IF;
END_REGION

REGION Network 14: If PID enabled, calculate heating target
   RUNG wire#powerrail
      Contact( "AI_PID_Bon4_Enable" )
      { S7_Templates := "SrcType := Real"; S7_GenerateENO := "TRUE" } Mul(in1 := "AI_PID_Bon4_CV", in2 := 0.95, out => "AI_TT3219_Bon4_Target")
   END_RUNG
   // the same network as SCL:
   IF "AI_PID_Bon4_Enable" THEN "AI_TT3219_Bon4_Target" := "AI_PID_Bon4_CV" * 0.95; END_IF;
END_REGION

REGION Network 15: If PID enabled, add ambient base to target
   RUNG wire#powerrail
      Contact( "AI_PID_Bon4_Enable" )
      { S7_Templates := "SrcType := Real"; S7_GenerateENO := "TRUE" } Add(in1 := "AI_TT3219_Bon4_Target", in2 := 25.0, out => "AI_TT3219_Bon4_Target")
   END_RUNG
   // the same network as SCL:
   IF "AI_PID_Bon4_Enable" THEN "AI_TT3219_Bon4_Target" := "AI_TT3219_Bon4_Target" + 25.0; END_IF;
END_REGION

REGION Network 16: If PID disabled, set target to ambient
   RUNG wire#powerrail
      I_Contact( "AI_PID_Bon4_Enable" )
      { S7_GenerateENO := "TRUE" } Move(in := 25.0, out1 => "AI_TT3219_Bon4_Target")
   END_RUNG
   // the same network as SCL:
   IF NOT "AI_PID_Bon4_Enable" THEN "AI_TT3219_Bon4_Target" := 25.0; END_IF;
END_REGION

REGION Network 17: Calculate memory term: Pure * 0.995
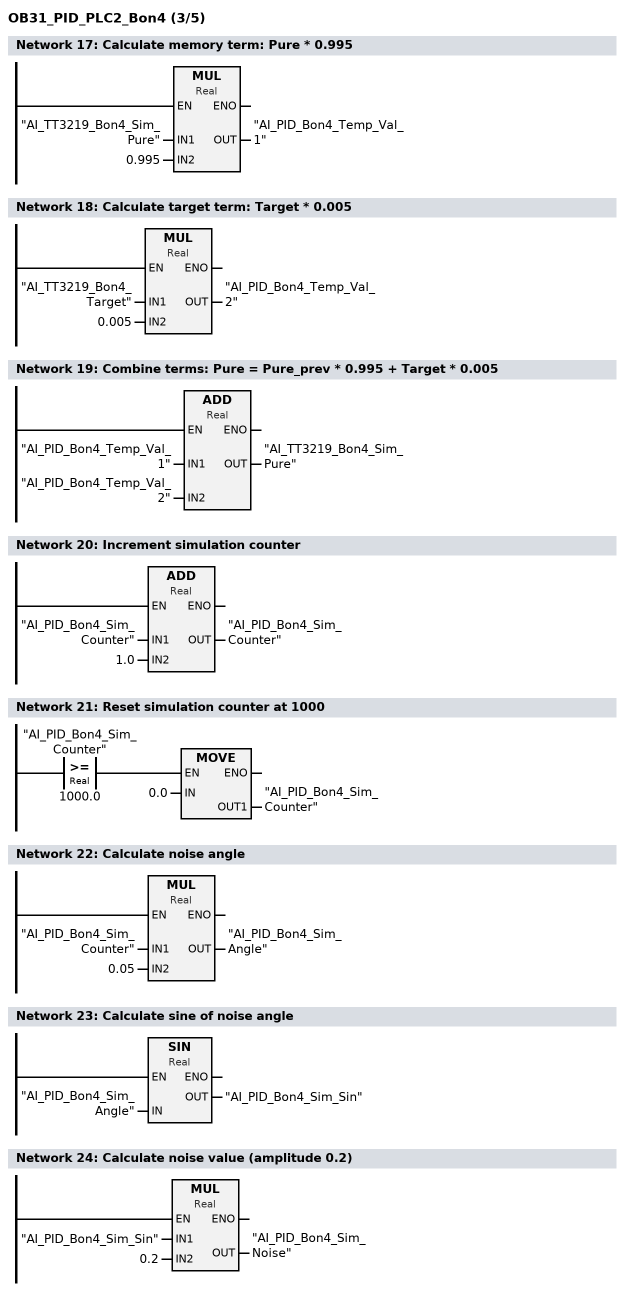
   RUNG wire#powerrail
      { S7_Templates := "SrcType := Real"; S7_GenerateENO := "TRUE" } Mul(in1 := "AI_TT3219_Bon4_Sim_Pure", in2 := 0.995, out => "AI_PID_Bon4_Temp_Val_1")
   END_RUNG
   // the same network as SCL:
   "AI_PID_Bon4_Temp_Val_1" := "AI_TT3219_Bon4_Sim_Pure" * 0.995;
END_REGION

REGION Network 18: Calculate target term: Target * 0.005
   RUNG wire#powerrail
      { S7_Templates := "SrcType := Real"; S7_GenerateENO := "TRUE" } Mul(in1 := "AI_TT3219_Bon4_Target", in2 := 0.005, out => "AI_PID_Bon4_Temp_Val_2")
   END_RUNG
   // the same network as SCL:
   "AI_PID_Bon4_Temp_Val_2" := "AI_TT3219_Bon4_Target" * 0.005;
END_REGION

REGION Network 19: Combine terms: Pure = Pure_prev * 0.995 + Target * 0.005
   RUNG wire#powerrail
      { S7_Templates := "SrcType := Real"; S7_GenerateENO := "TRUE" } Add(in1 := "AI_PID_Bon4_Temp_Val_1", in2 := "AI_PID_Bon4_Temp_Val_2", out => "AI_TT3219_Bon4_Sim_Pure")
   END_RUNG
   // the same network as SCL:
   "AI_TT3219_Bon4_Sim_Pure" := "AI_PID_Bon4_Temp_Val_1" + "AI_PID_Bon4_Temp_Val_2";
END_REGION

REGION Network 20: Increment simulation counter
   RUNG wire#powerrail
      { S7_Templates := "SrcType := Real"; S7_GenerateENO := "TRUE" } Add(in1 := "AI_PID_Bon4_Sim_Counter", in2 := 1.0, out => "AI_PID_Bon4_Sim_Counter")
   END_RUNG
   // the same network as SCL:
   "AI_PID_Bon4_Sim_Counter" := "AI_PID_Bon4_Sim_Counter" + 1.0;
END_REGION

REGION Network 21: Reset simulation counter at 1000
   RUNG wire#powerrail
      { S7_Templates := "SrcType := Real" } GE_Contact(in1 := "AI_PID_Bon4_Sim_Counter", in2 := 1000.0)
      { S7_GenerateENO := "TRUE" } Move(in := 0.0, out1 => "AI_PID_Bon4_Sim_Counter")
   END_RUNG
   // the same network as SCL:
   IF "AI_PID_Bon4_Sim_Counter" >= 1000.0 THEN "AI_PID_Bon4_Sim_Counter" := 0.0; END_IF;
END_REGION

REGION Network 22: Calculate noise angle
   RUNG wire#powerrail
      { S7_Templates := "SrcType := Real"; S7_GenerateENO := "TRUE" } Mul(in1 := "AI_PID_Bon4_Sim_Counter", in2 := 0.05, out => "AI_PID_Bon4_Sim_Angle")
   END_RUNG
   // the same network as SCL:
   "AI_PID_Bon4_Sim_Angle" := "AI_PID_Bon4_Sim_Counter" * 0.05;
END_REGION

REGION Network 23: Calculate sine of noise angle
   "AI_PID_Bon4_Sim_Sin" := SIN("AI_PID_Bon4_Sim_Angle");
END_REGION

REGION Network 24: Calculate noise value (amplitude 0.2)
   RUNG wire#powerrail
      { S7_Templates := "SrcType := Real"; S7_GenerateENO := "TRUE" } Mul(in1 := "AI_PID_Bon4_Sim_Sin", in2 := 0.2, out => "AI_PID_Bon4_Sim_Noise")
   END_RUNG
   // the same network as SCL:
   "AI_PID_Bon4_Sim_Noise" := "AI_PID_Bon4_Sim_Sin" * 0.2;
END_REGION

REGION Network 25: Add noise to pure temperature to get noisy PV
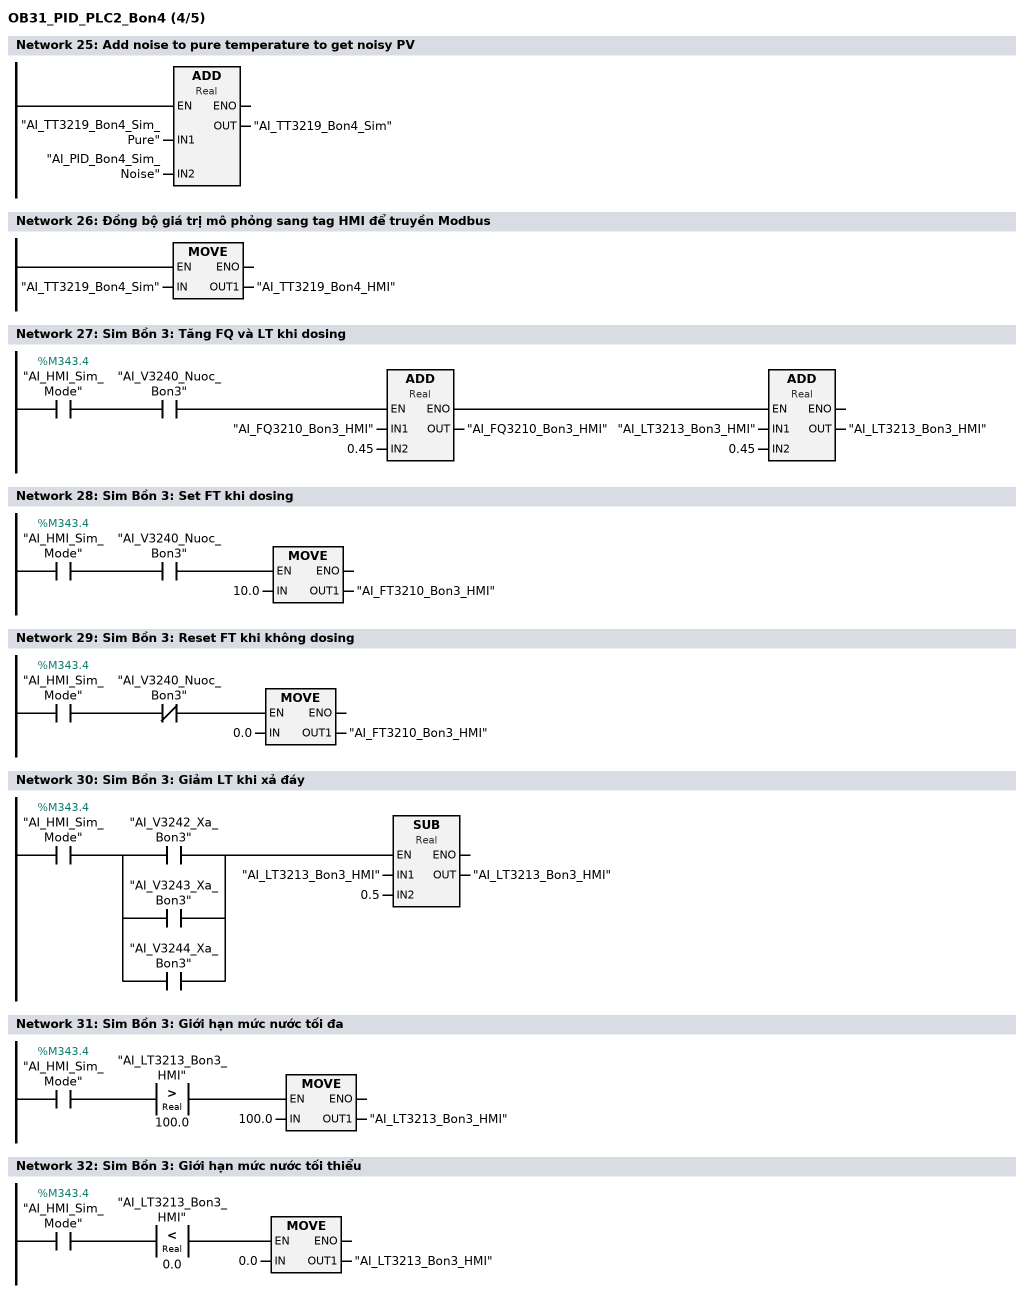
   RUNG wire#powerrail
      { S7_Templates := "SrcType := Real"; S7_GenerateENO := "TRUE" } Add(in1 := "AI_TT3219_Bon4_Sim_Pure", in2 := "AI_PID_Bon4_Sim_Noise", out => "AI_TT3219_Bon4_Sim")
   END_RUNG
   // the same network as SCL:
   "AI_TT3219_Bon4_Sim" := "AI_TT3219_Bon4_Sim_Pure" + "AI_PID_Bon4_Sim_Noise";
END_REGION

REGION Network 26: Đồng bộ giá trị mô phỏng sang tag HMI để truyền Modbus
   RUNG wire#powerrail
      { S7_GenerateENO := "TRUE" } Move(in := "AI_TT3219_Bon4_Sim", out1 => "AI_TT3219_Bon4_HMI")
   END_RUNG
   // the same network as SCL:
   "AI_TT3219_Bon4_HMI" := "AI_TT3219_Bon4_Sim";
END_REGION

REGION Network 27: Sim Bồn 3: Tăng FQ và LT khi dosing
   RUNG wire#powerrail
      Contact( "AI_HMI_Sim_Mode" )
      Contact( "AI_V3240_Nuoc_Bon3" )
      { S7_Templates := "SrcType := Real"; S7_GenerateENO := "TRUE" } Add(in1 := "AI_FQ3210_Bon3_HMI", in2 := 0.45, out => "AI_FQ3210_Bon3_HMI")
      { S7_Templates := "SrcType := Real"; S7_GenerateENO := "TRUE" } Add(in1 := "AI_LT3213_Bon3_HMI", in2 := 0.45, out => "AI_LT3213_Bon3_HMI")
   END_RUNG
   // the same network as SCL:
   // ENO of a box is taken as its EN; it also drops when the box reports an error
   IF "AI_HMI_Sim_Mode" AND "AI_V3240_Nuoc_Bon3" THEN
       "AI_FQ3210_Bon3_HMI" := "AI_FQ3210_Bon3_HMI" + 0.45;
       "AI_LT3213_Bon3_HMI" := "AI_LT3213_Bon3_HMI" + 0.45;
   END_IF;
END_REGION

REGION Network 28: Sim Bồn 3: Set FT khi dosing
   RUNG wire#powerrail
      Contact( "AI_HMI_Sim_Mode" )
      Contact( "AI_V3240_Nuoc_Bon3" )
      { S7_GenerateENO := "TRUE" } Move(in := 10.0, out1 => "AI_FT3210_Bon3_HMI")
   END_RUNG
   // the same network as SCL:
   IF "AI_HMI_Sim_Mode" AND "AI_V3240_Nuoc_Bon3" THEN "AI_FT3210_Bon3_HMI" := 10.0; END_IF;
END_REGION

REGION Network 29: Sim Bồn 3: Reset FT khi không dosing
   RUNG wire#powerrail
      Contact( "AI_HMI_Sim_Mode" )
      I_Contact( "AI_V3240_Nuoc_Bon3" )
      { S7_GenerateENO := "TRUE" } Move(in := 0.0, out1 => "AI_FT3210_Bon3_HMI")
   END_RUNG
   // the same network as SCL:
   IF "AI_HMI_Sim_Mode" AND NOT "AI_V3240_Nuoc_Bon3" THEN "AI_FT3210_Bon3_HMI" := 0.0; END_IF;
END_REGION

REGION Network 30: Sim Bồn 3: Giảm LT khi xả đáy
   RUNG wire#powerrail
      Contact( "AI_HMI_Sim_Mode" )
      wire#w1
      Contact( "AI_V3242_Xa_Bon3" )
      wire#w2
      { S7_Templates := "SrcType := Real"; S7_GenerateENO := "TRUE" } Sub(in1 := "AI_LT3213_Bon3_HMI", in2 := 0.5, out => "AI_LT3213_Bon3_HMI")
   END_RUNG
   RUNG wire#w1
      Contact( "AI_V3243_Xa_Bon3" )
   END_RUNG wire#w2
   RUNG wire#w1
      Contact( "AI_V3244_Xa_Bon3" )
   END_RUNG wire#w2
   // the same network as SCL:
   IF "AI_HMI_Sim_Mode" AND ("AI_V3242_Xa_Bon3" OR "AI_V3243_Xa_Bon3" OR "AI_V3244_Xa_Bon3") THEN
       "AI_LT3213_Bon3_HMI" := "AI_LT3213_Bon3_HMI" - 0.5;
   END_IF;
END_REGION

REGION Network 31: Sim Bồn 3: Giới hạn mức nước tối đa
   RUNG wire#powerrail
      Contact( "AI_HMI_Sim_Mode" )
      { S7_Templates := "SrcType := Real" } GT_Contact(in1 := "AI_LT3213_Bon3_HMI", in2 := 100.0)
      { S7_GenerateENO := "TRUE" } Move(in := 100.0, out1 => "AI_LT3213_Bon3_HMI")
   END_RUNG
   // the same network as SCL:
   IF "AI_HMI_Sim_Mode" AND ("AI_LT3213_Bon3_HMI" > 100.0) THEN "AI_LT3213_Bon3_HMI" := 100.0; END_IF;
END_REGION

